LIN {X 0,Y 154.357,Z 466.364,A -85,B 0,C 180,E1 -24102.965,E2 -24102.965} C_VEL
LIN {X 0,Y 157.924,Z 467.612,A -85,B 0,C 180,E1 -24108.246,E2 -24108.246} C_VEL
LIN {X 0,Y 162.729,Z 467.187,A -85,B 0,C 180,E1 -24113.367,E2 -24113.367} C_VEL
LIN {X 0,Y 167.861,Z 465.471,A -85,B 0,C 180,E1 -24117.601,E2 -24117.601} C_VEL
LIN {X 0,Y 173.217,Z 462.762,A -85,B 0,C 180,E1 -24121.163,E2 -24121.163} C_VEL
LIN {X 0,Y 179.055,Z 458.948,A -85,B 0,C 180,E1 -24124.503,E2 -24124.503} C_VEL
LIN {X 0,Y 186.333,Z 453.105,A -85,B 0,C 180,E1 -24128.018,E2 -24128.018} C_VEL
LIN {X 0,Y 187.702,Z 451.908,A -85,B 0,C 180,E1 -24128.614,E2 -24128.614} C_VEL
LIN {X 0,Y 189.446,Z 450.085,A -85,B 0,C 180,E1 -24129.61,E2 -24129.61} C_VEL
LIN {X 0,Y 191.01,Z 446.938,A -85,B 0,C 180,E1 -24132.754,E2 -24132.754} C_VEL
LIN {X 0,Y 191.797,Z 445.035,A -85,B 0,C 180,E1 -24134.863,E2 -24134.863} C_VEL
LIN {X 0,Y 192.282,Z 443.477,A -85,B 0,C 180,E1 -24137.002,E2 -24137.002} C_VEL
LIN {X 0,Y 192.219,Z 442.595,A -85,B 0,C 180,E1 -24139.212,E2 -24139.212} C_VEL
LIN {X 0,Y 191.954,Z 442.263,A -85,B 0,C 180,E1 -24141.477,E2 -24141.477} C_VEL
LIN {X 0,Y 191.608,Z 442.354,A -85,B 0,C 180,E1 -24143.795,E2 -24143.795} C_VEL
LIN {X 0,Y 191.277,Z 442.94,A -85,B 0,C 180,E1 -24146.162,E2 -24146.162} C_VEL
LIN {X 0,Y 190.853,Z 444.09,A -85,B 0,C 180,E1 -24148.602,E2 -24148.602} C_VEL
LIN {X 0,Y 190.613,Z 447.54,A -85,B 0,C 180,E1 -24153.577,E2 -24153.577} C_VEL
LIN {X 0,Y 190.373,Z 450.298,A -85,B 0,C 180,E1 -24156.205,E2 -24156.205} C_VEL
LIN {X 0,Y 189.792,Z 454.164,A -85,B 0,C 180,E1 -24159.014,E2 -24159.014} C_VEL
LIN {X 0,Y 188.189,Z 457.579,A -85,B 0,C 180,E1 -24160.569,E2 -24160.569} C_VEL
LIN {X 0,Y 184.271,Z 464.734,A -85,B 0,C 180,E1 -24163.562,E2 -24163.562} C_VEL
LIN {X 0,Y 178.792,Z 473.353,A -85,B 0,C 180,E1 -24167.309,E2 -24167.309} C_VEL
LIN {X 0,Y 173.001,Z 480.936,A -85,B 0,C 180,E1 -24170.975,E2 -24170.975} C_VEL
LIN {X 0,Y 166.298,Z 488.194,A -85,B 0,C 180,E1 -24175.214,E2 -24175.214} C_VEL
LIN {X 0,Y 160.237,Z 493.898,A -85,B 0,C 180,E1 -24179.71,E2 -24179.71} C_VEL
LIN {X 0,Y 156.331,Z 497.231,A -85,B 0,C 180,E1 -24183.285,E2 -24183.285} C_VEL
LIN {X 0,Y 152.307,Z 500.47,A -85,B 0,C 180,E1 -24188.337,E2 -24188.337} C_VEL
LIN {X 0,Y 149.986,Z 502.425,A -85,B 0,C 180,E1 -24193.672,E2 -24193.672} C_VEL
LIN {X 0,Y 149.209,Z 503.02,A -85,B 0,C 180,E1 -24199.14,E2 -24199.14} C_VEL
LIN {X 0,Y 149.908,Z 502.28,A -85,B 0,C 180,E1 -24204.62,E2 -24204.62} C_VEL
LIN {X 0,Y 150.705,Z 501.363,A -85,B 0,C 180,E1 -24207.327,E2 -24207.327} C_VEL
LIN {X 0,Y 151.499,Z 500.007,A -85,B 0,C 180,E1 -24210,E2 -24210} C_VEL
LIN {X 0,Y 150.756,Z 496.519,A -85,B 0,C 180,E1 -24214.01,E2 -24214.01} C_VEL
LIN {X 0,Y 150.197,Z 491.756,A -85,B 0,C 180,E1 -24218.069,E2 -24218.069} C_VEL
LIN {X 0,Y 150.286,Z 485.644,A -85,B 0,C 180,E1 -24222.148,E2 -24222.148} C_VEL
LIN {X 0,Y 151,Z 477.97,A -85,B 0,C 180,E1 -24226.216,E2 -24226.216} C_VEL
LIN {X 0,Y 152.213,Z 470.164,A -85,B 0,C 180,E1 -24229.557,E2 -24229.557} C_VEL
LIN {X 0,Y 152.227,Z 462.309,A -85,B 0,C 180,E1 -24232.318,E2 -24232.318} C_VEL
LIN {X 0,Y 152.281,Z 452.364,A -85,B 0,C 180,E1 -24235.27,E2 -24235.27} C_VEL
LIN {X 0,Y 152.315,Z 441.552,A -85,B 0,C 180,E1 -24237.914,E2 -24237.914} C_VEL
LIN {X 0,Y 152.221,Z 428.27,A -85,B 0,C 180,E1 -24240.521,E2 -24240.521} C_VEL
LIN {X 0,Y 152.051,Z 415.268,A -85,B 0,C 180,E1 -24242.501,E2 -24242.501} C_VEL
LIN {X 0,Y 151.716,Z 401.613,A -85,B 0,C 180,E1 -24244.059,E2 -24244.059} C_VEL
LIN {X 0,Y 151.32,Z 399.501,A -85,B 0,C 180,E1 -24244.647,E2 -24244.647} C_VEL
LIN {X 0,Y 150.434,Z 397.793,A -85,B 0,C 180,E1 -24245.814,E2 -24245.814} C_VEL
LIN {X 0,Y 146.596,Z 391.678,A -85,B 0,C 180,E1 -24251.674,E2 -24251.674} C_VEL
LIN {X 0,Y 145.381,Z 388.003,A -85,B 0,C 180,E1 -24254.938,E2 -24254.938} C_VEL
LIN {X 0,Y 144.009,Z 381.533,A -85,B 0,C 180,E1 -24261.336,E2 -24261.336} C_VEL
LIN {X 0,Y 143.314,Z 377.702,A -85,B 0,C 180,E1 -24265.393,E2 -24265.393} C_VEL
LIN {X 0,Y 143.186,Z 377.647,A -85,B 0,C 180,E1 -24272.064,E2 -24272.064} C_VEL
LIN {X 0,Y 143.264,Z 377.634,A -85,B 0,C 180,E1 -24278.756,E2 -24278.756} C_VEL
LIN {X 0,Y 143.264,Z 377.64,A -85,B 0,C 180,E1 -24282.882,E2 -24282.882} C_VEL
LIN {X 0,Y 143.53,Z 377.598,A -85,B 0,C 180,E1 -24288.705,E2 -24288.705} C_VEL
LIN {X 0,Y 143.618,Z 377.594,A -85,B 0,C 180,E1 -24291.558,E2 -24291.558} C_VEL
LIN {X 0,Y 144.171,Z 377.525,A -85,B 0,C 180,E1 -24300,E2 -24300} C_VEL
LIN {X 0,Y 143.656,Z 377.59,A -85,B 0,C 180,E1 -24308.44,E2 -24308.44} C_VEL
LIN {X 0,Y 143.545,Z 377.601,A -85,B 0,C 180,E1 -24311.713,E2 -24311.713} C_VEL
LIN {X 0,Y 143.302,Z 377.634,A -85,B 0,C 180,E1 -24317.113,E2 -24317.113} C_VEL
LIN {X 0,Y 143.274,Z 377.632,A -85,B 0,C 180,E1 -24321.255,E2 -24321.255} C_VEL
LIN {X 0,Y 143.188,Z 377.648,A -85,B 0,C 180,E1 -24327.938,E2 -24327.938} C_VEL
LIN {X 0,Y 143.167,Z 377.65,A -85,B 0,C 180,E1 -24333.436,E2 -24333.436} C_VEL
LIN {X 0,Y 143.077,Z 377.659,A -85,B 0,C 180,E1 -24339.685,E2 -24339.685} C_VEL
LIN {X 0,Y 143.066,Z 377.663,A -85,B 0,C 180,E1 -24343.451,E2 -24343.451} C_VEL
LIN {X 0,Y 143.069,Z 377.659,A -85,B 0,C 180,E1 -24347.464,E2 -24347.464} C_VEL
LIN {X 0,Y 143.106,Z 377.659,A -85,B 0,C 180,E1 -24351.792,E2 -24351.792} C_VEL
LIN {X 0,Y 143.185,Z 377.647,A -85,B 0,C 180,E1 -24357.323,E2 -24357.323} C_VEL
LIN {X 0,Y 143.191,Z 377.644,A -85,B 0,C 180,E1 -24362.063,E2 -24362.063} C_VEL
LIN {X 0,Y 143.278,Z 377.636,A -85,B 0,C 180,E1 -24368.746,E2 -24368.746} C_VEL
LIN {X 0,Y 143.318,Z 377.629,A -85,B 0,C 180,E1 -24372.889,E2 -24372.889} C_VEL
LIN {X 0,Y 143.604,Z 377.592,A -85,B 0,C 180,E1 -24378.711,E2 -24378.711} C_VEL
LIN {X 0,Y 143.687,Z 377.585,A -85,B 0,C 180,E1 -24381.562,E2 -24381.562} C_VEL
LIN {X 0,Y 144.18,Z 377.526,A -85,B 0,C 180,E1 -24390,E2 -24390} C_VEL
LIN {X 0,Y 143.662,Z 377.589,A -85,B 0,C 180,E1 -24398.439,E2 -24398.439} C_VEL
LIN {X 0,Y 143.549,Z 377.598,A -85,B 0,C 180,E1 -24401.712,E2 -24401.712} C_VEL
LIN {X 0,Y 143.309,Z 377.631,A -85,B 0,C 180,E1 -24407.112,E2 -24407.112} C_VEL
LIN {X 0,Y 143.279,Z 377.636,A -85,B 0,C 180,E1 -24411.255,E2 -24411.255} C_VEL
LIN {X 0,Y 143.204,Z 377.646,A -85,B 0,C 180,E1 -24418.433,E2 -24418.433} C_VEL
LIN {X 0,Y 143.215,Z 377.783,A -85,B 0,C 180,E1 -24419.148,E2 -24419.148} C_VEL
LIN {X 0,Y 143.551,Z 379.072,A -85,B 0,C 180,E1 -24419.715,E2 -24419.715} C_VEL
LIN {X 0,Y 147.266,Z 391.351,A -85,B 0,C 180,E1 -24422.471,E2 -24422.471} C_VEL
LIN {X 0,Y 150.191,Z 402.477,A -85,B 0,C 180,E1 -24425.295,E2 -24425.295} C_VEL
LIN {X 0,Y 151.278,Z 407.074,A -85,B 0,C 180,E1 -24426.585,E2 -24426.585} C_VEL
LIN {X 0,Y 150.775,Z 410.846,A -85,B 0,C 180,E1 -24427.589,E2 -24427.589} C_VEL
LIN {X 0,Y 148.66,Z 421.695,A -85,B 0,C 180,E1 -24430.851,E2 -24430.851} C_VEL
LIN {X 0,Y 146.664,Z 431.947,A -85,B 0,C 180,E1 -24434.715,E2 -24434.715} C_VEL
LIN {X 0,Y 145.272,Z 439.714,A -85,B 0,C 180,E1 -24438.302,E2 -24438.302} C_VEL
LIN {X 0,Y 144.152,Z 447.331,A -85,B 0,C 180,E1 -24442.593,E2 -24442.593} C_VEL
LIN {X 0,Y 143.579,Z 454.147,A -85,B 0,C 180,E1 -24447.423,E2 -24447.423} C_VEL
LIN {X 0,Y 143.684,Z 458.94,A -85,B 0,C 180,E1 -24451.692,E2 -24451.692} C_VEL
LIN {X 0,Y 144.77,Z 463.725,A -85,B 0,C 180,E1 -24457.272,E2 -24457.272} C_VEL
LIN {X 0,Y 147.105,Z 466.924,A -85,B 0,C 180,E1 -24462.84,E2 -24462.84} C_VEL
LIN {X 0,Y 150.694,Z 468.63,A -85,B 0,C 180,E1 -24468.34,E2 -24468.34} C_VEL
LIN {X 0,Y 155.575,Z 468.704,A -85,B 0,C 180,E1 -24473.621,E2 -24473.621} C_VEL
LIN {X 0,Y 161.684,Z 467.121,A -85,B 0,C 180,E1 -24478.668,E2 -24478.668} C_VEL
LIN {X 0,Y 168.951,Z 463.815,A -85,B 0,C 180,E1 -24483.318,E2 -24483.318} C_VEL
LIN {X 0,Y 175.778,Z 459.555,A -85,B 0,C 180,E1 -24486.889,E2 -24486.889} C_VEL
LIN {X 0,Y 182.642,Z 454.306,A -85,B 0,C 180,E1 -24489.972,E2 -24489.972} C_VEL
LIN {X 0,Y 184.158,Z 452.844,A -85,B 0,C 180,E1 -24491,E2 -24491} C_VEL
LIN {X 0,Y 185.308,Z 451.011,A -85,B 0,C 180,E1 -24493.153,E2 -24493.153} C_VEL
LIN {X 0,Y 186.297,Z 449.275,A -85,B 0,C 180,E1 -24495.312,E2 -24495.312} C_VEL
LIN {X 0,Y 186.916,Z 447.95,A -85,B 0,C 180,E1 -24497.506,E2 -24497.506} C_VEL
LIN {X 0,Y 186.882,Z 447.289,A -85,B 0,C 180,E1 -24499.925,E2 -24499.925} C_VEL
LIN {X 0,Y 186.707,Z 447.179,A -85,B 0,C 180,E1 -24502.112,E2 -24502.112} C_VEL
LIN {X 0,Y 186.317,Z 447.696,A -85,B 0,C 180,E1 -24505.14,E2 -24505.14} C_VEL
LIN {X 0,Y 186.072,Z 448.315,A -85,B 0,C 180,E1 -24506.952,E2 -24506.952} C_VEL
LIN {X 0,Y 185.445,Z 451.37,A -85,B 0,C 180,E1 -24512.044,E2 -24512.044} C_VEL
LIN {X 0,Y 185.308,Z 453.622,A -85,B 0,C 180,E1 -24514.673,E2 -24514.673} C_VEL
LIN {X 0,Y 184.592,Z 457.005,A -85,B 0,C 180,E1 -24517.53,E2 -24517.53} C_VEL
LIN {X 0,Y 184.039,Z 458.562,A -85,B 0,C 180,E1 -24518.509,E2 -24518.509} C_VEL
LIN {X 0,Y 179.381,Z 465.993,A -85,B 0,C 180,E1 -24521.894,E2 -24521.894} C_VEL
LIN {X 0,Y 174.417,Z 473.037,A -85,B 0,C 180,E1 -24525.16,E2 -24525.16} C_VEL
LIN {X 0,Y 169.27,Z 479.371,A -85,B 0,C 180,E1 -24528.372,E2 -24528.372} C_VEL
LIN {X 0,Y 163.931,Z 484.915,A -85,B 0,C 180,E1 -24531.565,E2 -24531.565} C_VEL
LIN {X 0,Y 157.251,Z 491.061,A -85,B 0,C 180,E1 -24536.038,E2 -24536.038} C_VEL
LIN {X 0,Y 152.664,Z 494.674,A -85,B 0,C 180,E1 -24539.577,E2 -24539.577} C_VEL
LIN {X 0,Y 147.621,Z 498.32,A -85,B 0,C 180,E1 -24544.63,E2 -24544.63} C_VEL
LIN {X 0,Y 144.256,Z 500.64,A -85,B 0,C 180,E1 -24550.061,E2 -24550.061} C_VEL
LIN {X 0,Y 142.518,Z 501.685,A -85,B 0,C 180,E1 -24555.726,E2 -24555.726} C_VEL
LIN {X 0,Y 142.435,Z 501.436,A -85,B 0,C 180,E1 -24561.488,E2 -24561.488} C_VEL
LIN {X 0,Y 143.727,Z 499.805,A -85,B 0,C 180,E1 -24567.197,E2 -24567.197} C_VEL
LIN {X 0,Y 144.54,Z 498.311,A -85,B 0,C 180,E1 -24570,E2 -24570} C_VEL
LIN {X 0,Y 143.749,Z 494.605,A -85,B 0,C 180,E1 -24574.206,E2 -24574.206} C_VEL
LIN {X 0,Y 143.219,Z 489.598,A -85,B 0,C 180,E1 -24578.465,E2 -24578.465} C_VEL
LIN {X 0,Y 143.379,Z 483.237,A -85,B 0,C 180,E1 -24582.743,E2 -24582.743} C_VEL
LIN {X 0,Y 144.239,Z 475.28,A -85,B 0,C 180,E1 -24586.998,E2 -24586.998} C_VEL
LIN {X 0,Y 145.174,Z 468.85,A -85,B 0,C 180,E1 -24589.808,E2 -24589.808} C_VEL
LIN {X 0,Y 145.165,Z 459.805,A -85,B 0,C 180,E1 -24593.093,E2 -24593.093} C_VEL
LIN {X 0,Y 145.254,Z 448,A -85,B 0,C 180,E1 -24596.586,E2 -24596.586} C_VEL
LIN {X 0,Y 145.302,Z 435.99,A -85,B 0,C 180,E1 -24599.468,E2 -24599.468} C_VEL
LIN {X 0,Y 145.193,Z 422.691,A -85,B 0,C 180,E1 -24601.982,E2 -24601.982} C_VEL
LIN {X 0,Y 145.003,Z 408.799,A -85,B 0,C 180,E1 -24603.987,E2 -24603.987} C_VEL
LIN {X 0,Y 144.923,Z 398.818,A -85,B 0,C 180,E1 -24605.188,E2 -24605.188} C_VEL
LIN {X 0,Y 146.169,Z 394.703,A -85,B 0,C 180,E1 -24608.685,E2 -24608.685} C_VEL
LIN {X 0,Y 146.437,Z 392.265,A -85,B 0,C 180,E1 -24610.919,E2 -24610.919} C_VEL
LIN {X 0,Y 145.381,Z 388.003,A -85,B 0,C 180,E1 -24614.938,E2 -24614.938} C_VEL
LIN {X 0,Y 144.38,Z 386.609,A -85,B 0,C 180,E1 -24616.344,E2 -24616.344} C_VEL
LIN {X 0,Y 141.069,Z 384.674,A -85,B 0,C 180,E1 -24618.55,E2 -24618.55} C_VEL
LIN {X 0,Y 137.744,Z 382.744,A -85,B 0,C 180,E1 -24620.858,E2 -24620.858} C_VEL
LIN {X 0,Y 136.779,Z 381.393,A -85,B 0,C 180,E1 -24622.388,E2 -24622.388} C_VEL
LIN {X 0,Y 136.26,Z 378.572,A -85,B 0,C 180,E1 -24625.611,E2 -24625.611} C_VEL
LIN {X 0,Y 136.142,Z 378.524,A -85,B 0,C 180,E1 -24632.315,E2 -24632.315} C_VEL
LIN {X 0,Y 136.231,Z 378.51,A -85,B 0,C 180,E1 -24638.831,E2 -24638.831} C_VEL
LIN {X 0,Y 136.23,Z 378.508,A -85,B 0,C 180,E1 -24645.052,E2 -24645.052} C_VEL
LIN {X 0,Y 136.423,Z 378.482,A -85,B 0,C 180,E1 -24648.177,E2 -24648.177} C_VEL
LIN {X 0,Y 136.544,Z 378.476,A -85,B 0,C 180,E1 -24651.117,E2 -24651.117} C_VEL
LIN {X 0,Y 137.128,Z 378.402,A -85,B 0,C 180,E1 -24660,E2 -24660} C_VEL
LIN {X 0,Y 136.584,Z 378.472,A -85,B 0,C 180,E1 -24668.88,E2 -24668.88} C_VEL
LIN {X 0,Y 136.489,Z 378.481,A -85,B 0,C 180,E1 -24671.955,E2 -24671.955} C_VEL
LIN {X 0,Y 136.241,Z 378.514,A -85,B 0,C 180,E1 -24678.03,E2 -24678.03} C_VEL
LIN {X 0,Y 136.195,Z 378.513,A -85,B 0,C 180,E1 -24681.749,E2 -24681.749} C_VEL
LIN {X 0,Y 136.098,Z 378.528,A -85,B 0,C 180,E1 -24688.617,E2 -24688.617} C_VEL
LIN {X 0,Y 136.077,Z 378.534,A -85,B 0,C 180,E1 -24694.619,E2 -24694.619} C_VEL
LIN {X 0,Y 136.052,Z 378.533,A -85,B 0,C 180,E1 -24699.21,E2 -24699.21} C_VEL
LIN {X 0,Y 136.006,Z 378.543,A -85,B 0,C 180,E1 -24703.662,E2 -24703.662} C_VEL
LIN {X 0,Y 136.033,Z 378.536,A -85,B 0,C 180,E1 -24707.808,E2 -24707.808} C_VEL
LIN {X 0,Y 136.055,Z 378.537,A -85,B 0,C 180,E1 -24711.695,E2 -24711.695} C_VEL
LIN {X 0,Y 136.09,Z 378.528,A -85,B 0,C 180,E1 -24715.718,E2 -24715.718} C_VEL
LIN {X 0,Y 136.147,Z 378.52,A -85,B 0,C 180,E1 -24722.317,E2 -24722.317} C_VEL
LIN {X 0,Y 136.245,Z 378.512,A -85,B 0,C 180,E1 -24728.834,E2 -24728.834} C_VEL
LIN {X 0,Y 136.287,Z 378.508,A -85,B 0,C 180,E1 -24735.059,E2 -24735.059} C_VEL
LIN {X 0,Y 136.502,Z 378.477,A -85,B 0,C 180,E1 -24738.115,E2 -24738.115} C_VEL
LIN {X 0,Y 136.61,Z 378.464,A -85,B 0,C 180,E1 -24741.122,E2 -24741.122} C_VEL
LIN {X 0,Y 137.137,Z 378.403,A -85,B 0,C 180,E1 -24750,E2 -24750} C_VEL
LIN {X 0,Y 136.59,Z 378.471,A -85,B 0,C 180,E1 -24758.879,E2 -24758.879} C_VEL
LIN {X 0,Y 136.492,Z 378.476,A -85,B 0,C 180,E1 -24761.954,E2 -24761.954} C_VEL
LIN {X 0,Y 136.248,Z 378.513,A -85,B 0,C 180,E1 -24768.028,E2 -24768.028} C_VEL
LIN {X 0,Y 136.2,Z 378.519,A -85,B 0,C 180,E1 -24771.749,E2 -24771.749} C_VEL
LIN {X 0,Y 136.215,Z 378.742,A -85,B 0,C 180,E1 -24778.366,E2 -24778.366} C_VEL
LIN {X 0,Y 136.564,Z 380.219,A -85,B 0,C 180,E1 -24778.952,E2 -24778.952} C_VEL
LIN {X 0,Y 140.044,Z 391.581,A -85,B 0,C 180,E1 -24781.629,E2 -24781.629} C_VEL
LIN {X 0,Y 142.86,Z 402.224,A -85,B 0,C 180,E1 -24784.453,E2 -24784.453} C_VEL
LIN {X 0,Y 144.294,Z 408.184,A -85,B 0,C 180,E1 -24786.195,E2 -24786.195} C_VEL
LIN {X 0,Y 142.369,Z 418.599,A -85,B 0,C 180,E1 -24789.244,E2 -24789.244} C_VEL
LIN {X 0,Y 140.108,Z 429.837,A -85,B 0,C 180,E1 -24793.338,E2 -24793.338} C_VEL
LIN {X 0,Y 138.322,Z 439.282,A -85,B 0,C 180,E1 -24797.684,E2 -24797.684} C_VEL
LIN {X 0,Y 137.152,Z 446.946,A -85,B 0,C 180,E1 -24802.055,E2 -24802.055} C_VEL
LIN {X 0,Y 136.487,Z 454.243,A -85,B 0,C 180,E1 -24807.271,E2 -24807.271} C_VEL
LIN {X 0,Y 136.663,Z 459.872,A -85,B 0,C 180,E1 -24812.43,E2 -24812.43} C_VEL
LIN {X 0,Y 137.548,Z 463.697,A -85,B 0,C 180,E1 -24816.88,E2 -24816.88} C_VEL
LIN {X 0,Y 139.85,Z 467.374,A -85,B 0,C 180,E1 -24822.707,E2 -24822.707} C_VEL
LIN {X 0,Y 143.461,Z 469.494,A -85,B 0,C 180,E1 -24828.45,E2 -24828.45} C_VEL
LIN {X 0,Y 146.201,Z 470.045,A -85,B 0,C 180,E1 -24831.708,E2 -24831.708} C_VEL
LIN {X 0,Y 149.094,Z 470.03,A -85,B 0,C 180,E1 -24834.59,E2 -24834.59} C_VEL
LIN {X 0,Y 154.629,Z 469.025,A -85,B 0,C 180,E1 -24839.143,E2 -24839.143} C_VEL
LIN {X 0,Y 162.013,Z 466.324,A -85,B 0,C 180,E1 -24843.888,E2 -24843.888} C_VEL
LIN {X 0,Y 168.225,Z 463.079,A -85,B 0,C 180,E1 -24847.2,E2 -24847.2} C_VEL
LIN {X 0,Y 175.256,Z 458.564,A -85,B 0,C 180,E1 -24850.396,E2 -24850.396} C_VEL
LIN {X 0,Y 177.687,Z 456.802,A -85,B 0,C 180,E1 -24851.406,E2 -24851.406} C_VEL
LIN {X 0,Y 179.485,Z 454.864,A -85,B 0,C 180,E1 -24853.588,E2 -24853.588} C_VEL
LIN {X 0,Y 180.701,Z 453.339,A -85,B 0,C 180,E1 -24855.798,E2 -24855.798} C_VEL
LIN {X 0,Y 181.365,Z 452.239,A -85,B 0,C 180,E1 -24858.06,E2 -24858.06} C_VEL
LIN {X 0,Y 181.364,Z 451.826,A -85,B 0,C 180,E1 -24861.566,E2 -24861.566} C_VEL
LIN {X 0,Y 180.963,Z 452.486,A -85,B 0,C 180,E1 -24865.29,E2 -24865.29} C_VEL
LIN {X 0,Y 180.506,Z 453.579,A -85,B 0,C 180,E1 -24867.854,E2 -24867.854} C_VEL
LIN {X 0,Y 180.026,Z 456.917,A -85,B 0,C 180,E1 -24873.13,E2 -24873.13} C_VEL
LIN {X 0,Y 179.314,Z 459.81,A -85,B 0,C 180,E1 -24876.009,E2 -24876.009} C_VEL
LIN {X 0,Y 178.876,Z 461.072,A -85,B 0,C 180,E1 -24877.004,E2 -24877.004} C_VEL
LIN {X 0,Y 177.22,Z 463.734,A -85,B 0,C 180,E1 -24878.446,E2 -24878.446} C_VEL
LIN {X 0,Y 172.055,Z 470.575,A -85,B 0,C 180,E1 -24881.802,E2 -24881.802} C_VEL
LIN {X 0,Y 165.796,Z 477.898,A -85,B 0,C 180,E1 -24885.621,E2 -24885.621} C_VEL
LIN {X 0,Y 160.266,Z 483.373,A -85,B 0,C 180,E1 -24888.87,E2 -24888.87} C_VEL
LIN {X 0,Y 153.015,Z 489.519,A -85,B 0,C 180,E1 -24893.339,E2 -24893.339} C_VEL
LIN {X 0,Y 146.557,Z 494.203,A -85,B 0,C 180,E1 -24898.165,E2 -24898.165} C_VEL
LIN {X 0,Y 141.21,Z 497.544,A -85,B 0,C 180,E1 -24903.39,E2 -24903.39} C_VEL
LIN {X 0,Y 137.573,Z 499.634,A -85,B 0,C 180,E1 -24909.048,E2 -24909.048} C_VEL
LIN {X 0,Y 135.637,Z 500.465,A -85,B 0,C 180,E1 -24914.985,E2 -24914.985} C_VEL
LIN {X 0,Y 135.44,Z 499.99,A -85,B 0,C 180,E1 -24921.045,E2 -24921.045} C_VEL
LIN {X 0,Y 136.769,Z 498.123,A -85,B 0,C 180,E1 -24927.055,E2 -24927.055} C_VEL
LIN {X 0,Y 137.592,Z 496.559,A -85,B 0,C 180,E1 -24930,E2 -24930} C_VEL
LIN {X 0,Y 136.729,Z 492.653,A -85,B 0,C 180,E1 -24934.422,E2 -24934.422} C_VEL
LIN {X 0,Y 136.239,Z 487.441,A -85,B 0,C 180,E1 -24938.903,E2 -24938.903} C_VEL
LIN {X 0,Y 136.45,Z 480.782,A -85,B 0,C 180,E1 -24943.401,E2 -24943.401} C_VEL
LIN {X 0,Y 137.524,Z 472.475,A -85,B 0,C 180,E1 -24947.855,E2 -24947.855} C_VEL
LIN {X 0,Y 138.132,Z 467.508,A -85,B 0,C 180,E1 -24950.086,E2 -24950.086} C_VEL
LIN {X 0,Y 138.079,Z 456.924,A -85,B 0,C 180,E1 -24954.028,E2 -24954.028} C_VEL
LIN {X 0,Y 138.187,Z 444.955,A -85,B 0,C 180,E1 -24957.65,E2 -24957.65} C_VEL
LIN {X 0,Y 138.258,Z 432.958,A -85,B 0,C 180,E1 -24960.551,E2 -24960.551} C_VEL
LIN {X 0,Y 138.262,Z 419.62,A -85,B 0,C 180,E1 -24963.122,E2 -24963.122} C_VEL
LIN {X 0,Y 138.102,Z 405.043,A -85,B 0,C 180,E1 -24965.212,E2 -24965.212} C_VEL
LIN {X 0,Y 138.081,Z 397.764,A -85,B 0,C 180,E1 -24966.14,E2 -24966.14} C_VEL
LIN {X 0,Y 139.151,Z 394.496,A -85,B 0,C 180,E1 -24969.086,E2 -24969.086} C_VEL
LIN {X 0,Y 139.317,Z 392.541,A -85,B 0,C 180,E1 -24970.979,E2 -24970.979} C_VEL
LIN {X 0,Y 137.852,Z 386.623,A -85,B 0,C 180,E1 -24976.893,E2 -24976.893} C_VEL
LIN {X 0,Y 136.779,Z 381.393,A -85,B 0,C 180,E1 -24982.388,E2 -24982.388} C_VEL
LIN {X 0,Y 136.203,Z 380.228,A -85,B 0,C 180,E1 -24983.939,E2 -24983.939} C_VEL
LIN {X 0,Y 134.584,Z 379.264,A -85,B 0,C 180,E1 -24986.31,E2 -24986.31} C_VEL
LIN {X 0,Y 132.573,Z 378.987,A -85,B 0,C 180,E1 -24988.714,E2 -24988.714} C_VEL
LIN {X 0,Y 129.287,Z 379.385,A -85,B 0,C 180,E1 -24993.846,E2 -24993.846} C_VEL
LIN {X 0,Y 129.002,Z 379.405,A -85,B 0,C 180,E1 -24995.637,E2 -24995.637} C_VEL
LIN {X 0,Y 129.111,Z 379.402,A -85,B 0,C 180,E1 -25000.937,E2 -25000.937} C_VEL
LIN {X 0,Y 129.341,Z 379.364,A -85,B 0,C 180,E1 -25007.97,E2 -25007.97} C_VEL
LIN {X 0,Y 129.467,Z 379.355,A -85,B 0,C 180,E1 -25010.627,E2 -25010.627} C_VEL
LIN {X 0,Y 130.083,Z 379.28,A -85,B 0,C 180,E1 -25020,E2 -25020} C_VEL
LIN {X 0,Y 129.511,Z 379.352,A -85,B 0,C 180,E1 -25029.369,E2 -25029.369} C_VEL
LIN {X 0,Y 129.39,Z 379.363,A -85,B 0,C 180,E1 -25032.548,E2 -25032.548} C_VEL
LIN {X 0,Y 129.152,Z 379.396,A -85,B 0,C 180,E1 -25039.056,E2 -25039.056} C_VEL
LIN {X 0,Y 129.106,Z 379.397,A -85,B 0,C 180,E1 -25042.399,E2 -25042.399} C_VEL
LIN {X 0,Y 129.034,Z 379.406,A -85,B 0,C 180,E1 -25049.374,E2 -25049.374} C_VEL
LIN {X 0,Y 128.991,Z 379.416,A -85,B 0,C 180,E1 -25055.19,E2 -25055.19} C_VEL
LIN {X 0,Y 128.975,Z 379.418,A -85,B 0,C 180,E1 -25060.836,E2 -25060.836} C_VEL
LIN {X 0,Y 128.924,Z 379.422,A -85,B 0,C 180,E1 -25065.126,E2 -25065.126} C_VEL
LIN {X 0,Y 128.957,Z 379.421,A -85,B 0,C 180,E1 -25069.728,E2 -25069.728} C_VEL
LIN {X 0,Y 128.991,Z 379.411,A -85,B 0,C 180,E1 -25074.812,E2 -25074.812} C_VEL
LIN {X 0,Y 129.051,Z 379.408,A -85,B 0,C 180,E1 -25080.652,E2 -25080.652} C_VEL
LIN {X 0,Y 129.108,Z 379.404,A -85,B 0,C 180,E1 -25087.728,E2 -25087.728} C_VEL
LIN {X 0,Y 129.161,Z 379.39,A -85,B 0,C 180,E1 -25090.945,E2 -25090.945} C_VEL
LIN {X 0,Y 129.42,Z 379.361,A -85,B 0,C 180,E1 -25097.816,E2 -25097.816} C_VEL
LIN {X 0,Y 129.532,Z 379.345,A -85,B 0,C 180,E1 -25100.633,E2 -25100.633} C_VEL
LIN {X 0,Y 130.092,Z 379.281,A -85,B 0,C 180,E1 -25110,E2 -25110} C_VEL
LIN {X 0,Y 129.516,Z 379.353,A -85,B 0,C 180,E1 -25119.369,E2 -25119.369} C_VEL
LIN {X 0,Y 129.394,Z 379.361,A -85,B 0,C 180,E1 -25122.548,E2 -25122.548} C_VEL
LIN {X 0,Y 129.158,Z 379.398,A -85,B 0,C 180,E1 -25129.055,E2 -25129.055} C_VEL
LIN {X 0,Y 129.109,Z 379.403,A -85,B 0,C 180,E1 -25132.398,E2 -25132.398} C_VEL
LIN {X 0,Y 129.111,Z 379.513,A -85,B 0,C 180,E1 -25137.34,E2 -25137.34} C_VEL
LIN {X 0,Y 129.362,Z 380.61,A -85,B 0,C 180,E1 -25137.942,E2 -25137.942} C_VEL
LIN {X 0,Y 132.87,Z 392.094,A -85,B 0,C 180,E1 -25140.777,E2 -25140.777} C_VEL
LIN {X 0,Y 135.839,Z 403.192,A -85,B 0,C 180,E1 -25143.881,E2 -25143.881} C_VEL
LIN {X 0,Y 137.231,Z 408.847,A -85,B 0,C 180,E1 -25145.629,E2 -25145.629} C_VEL
LIN {X 0,Y 135.513,Z 418.313,A -85,B 0,C 180,E1 -25148.487,E2 -25148.487} C_VEL
LIN {X 0,Y 133.301,Z 428.928,A -85,B 0,C 180,E1 -25152.429,E2 -25152.429} C_VEL
LIN {X 0,Y 131.445,Z 438.503,A -85,B 0,C 180,E1 -25156.885,E2 -25156.885} C_VEL
LIN {X 0,Y 130.136,Z 446.657,A -85,B 0,C 180,E1 -25161.607,E2 -25161.607} C_VEL
LIN {X 0,Y 129.396,Z 454.227,A -85,B 0,C 180,E1 -25167.102,E2 -25167.102} C_VEL
LIN {X 0,Y 129.598,Z 460.172,A -85,B 0,C 180,E1 -25172.552,E2 -25172.552} C_VEL
LIN {X 0,Y 130.703,Z 464.645,A -85,B 0,C 180,E1 -25177.889,E2 -25177.889} C_VEL
LIN {X 0,Y 132.578,Z 467.655,A -85,B 0,C 180,E1 -25182.585,E2 -25182.585} C_VEL
LIN {X 0,Y 136.224,Z 470.238,A -85,B 0,C 180,E1 -25188.582,E2 -25188.582} C_VEL
LIN {X 0,Y 138.346,Z 470.922,A -85,B 0,C 180,E1 -25191.234,E2 -25191.234} C_VEL
LIN {X 0,Y 141.253,Z 471.297,A -85,B 0,C 180,E1 -25194.309,E2 -25194.309} C_VEL
LIN {X 0,Y 147.586,Z 470.778,A -85,B 0,C 180,E1 -25199.694,E2 -25199.694} C_VEL
LIN {X 0,Y 155.102,Z 468.626,A -85,B 0,C 180,E1 -25204.557,E2 -25204.557} C_VEL
LIN {X 0,Y 160.575,Z 466.351,A -85,B 0,C 180,E1 -25207.545,E2 -25207.545} C_VEL
LIN {X 0,Y 167.851,Z 462.44,A -85,B 0,C 180,E1 -25210.861,E2 -25210.861} C_VEL
LIN {X 0,Y 172.473,Z 459.413,A -85,B 0,C 180,E1 -25212.951,E2 -25212.951} C_VEL
LIN {X 0,Y 173.501,Z 458.564,A -85,B 0,C 180,E1 -25214.066,E2 -25214.066} C_VEL
LIN {X 0,Y 174.968,Z 457.191,A -85,B 0,C 180,E1 -25216.33,E2 -25216.33} C_VEL
LIN {X 0,Y 175.649,Z 456.336,A -85,B 0,C 180,E1 -25218.669,E2 -25218.669} C_VEL
LIN {X 0,Y 175.803,Z 456.179,A -85,B 0,C 180,E1 -25221.087,E2 -25221.087} C_VEL
LIN {X 0,Y 175.516,Z 456.527,A -85,B 0,C 180,E1 -25223.605,E2 -25223.605} C_VEL
LIN {X 0,Y 175.288,Z 457.266,A -85,B 0,C 180,E1 -25226.17,E2 -25226.17} C_VEL
LIN {X 0,Y 174.39,Z 460.669,A -85,B 0,C 180,E1 -25232.19,E2 -25232.19} C_VEL
LIN {X 0,Y 173.947,Z 462.597,A -85,B 0,C 180,E1 -25234.447,E2 -25234.447} C_VEL
LIN {X 0,Y 173.375,Z 464.096,A -85,B 0,C 180,E1 -25235.835,E2 -25235.835} C_VEL
LIN {X 0,Y 172.76,Z 465.1,A -85,B 0,C 180,E1 -25236.542,E2 -25236.542} C_VEL
LIN {X 0,Y 167.757,Z 471.028,A -85,B 0,C 180,E1 -25239.691,E2 -25239.691} C_VEL
LIN {X 0,Y 160.732,Z 478.381,A -85,B 0,C 180,E1 -25243.826,E2 -25243.826} C_VEL
LIN {X 0,Y 154.939,Z 483.579,A -85,B 0,C 180,E1 -25247.127,E2 -25247.127} C_VEL
LIN {X 0,Y 147.332,Z 489.304,A -85,B 0,C 180,E1 -25251.676,E2 -25251.676} C_VEL
LIN {X 0,Y 140.557,Z 493.694,A -85,B 0,C 180,E1 -25256.633,E2 -25256.633} C_VEL
LIN {X 0,Y 134.881,Z 496.778,A -85,B 0,C 180,E1 -25262.035,E2 -25262.035} C_VEL
LIN {X 0,Y 130.941,Z 498.583,A -85,B 0,C 180,E1 -25267.932,E2 -25267.932} C_VEL
LIN {X 0,Y 128.807,Z 499.152,A -85,B 0,C 180,E1 -25274.169,E2 -25274.169} C_VEL
LIN {X 0,Y 128.483,Z 498.47,A -85,B 0,C 180,E1 -25280.555,E2 -25280.555} C_VEL
LIN {X 0,Y 129.799,Z 496.447,A -85,B 0,C 180,E1 -25286.896,E2 -25286.896} C_VEL
LIN {X 0,Y 130.652,Z 494.75,A -85,B 0,C 180,E1 -25290,E2 -25290} C_VEL
LIN {X 0,Y 129.717,Z 490.585,A -85,B 0,C 180,E1 -25294.661,E2 -25294.661} C_VEL
LIN {X 0,Y 129.335,Z 483.917,A -85,B 0,C 180,E1 -25300.289,E2 -25300.289} C_VEL
LIN {X 0,Y 129.734,Z 476.887,A -85,B 0,C 180,E1 -25304.911,E2 -25304.911} C_VEL
LIN {X 0,Y 131.014,Z 467.886,A -85,B 0,C 180,E1 -25309.588,E2 -25309.588} C_VEL
LIN {X 0,Y 131.012,Z 458.674,A -85,B 0,C 180,E1 -25313.377,E2 -25313.377} C_VEL
LIN {X 0,Y 131.107,Z 447.608,A -85,B 0,C 180,E1 -25317.105,E2 -25317.105} C_VEL
LIN {X 0,Y 131.235,Z 436.153,A -85,B 0,C 180,E1 -25320.243,E2 -25320.243} C_VEL
LIN {X 0,Y 131.282,Z 423.415,A -85,B 0,C 180,E1 -25323.049,E2 -25323.049} C_VEL
LIN {X 0,Y 131.258,Z 409.622,A -85,B 0,C 180,E1 -25325.375,E2 -25325.375} C_VEL
LIN {X 0,Y 131.229,Z 396.947,A -85,B 0,C 180,E1 -25327.068,E2 -25327.068} C_VEL
LIN {X 0,Y 132.112,Z 394.088,A -85,B 0,C 180,E1 -25329.669,E2 -25329.669} C_VEL
LIN {X 0,Y 131.992,Z 392.014,A -85,B 0,C 180,E1 -25331.803,E2 -25331.803} C_VEL
LIN {X 0,Y 130.636,Z 386.584,A -85,B 0,C 180,E1 -25337.554,E2 -25337.554} C_VEL
LIN {X 0,Y 129.584,Z 381.372,A -85,B 0,C 180,E1 -25343.374,E2 -25343.374} C_VEL
LIN {X 0,Y 129.186,Z 379.445,A -85,B 0,C 180,E1 -25345.785,E2 -25345.785} C_VEL
LIN {X 0,Y 129.049,Z 379.406,A -85,B 0,C 180,E1 -25350.65,E2 -25350.65} C_VEL
LIN {X 0,Y 129.002,Z 379.405,A -85,B 0,C 180,E1 -25355.637,E2 -25355.637} C_VEL
LIN {X 0,Y 128.367,Z 379.489,A -85,B 0,C 180,E1 -25358.242,E2 -25358.242} C_VEL
LIN {X 0,Y 126.825,Z 379.687,A -85,B 0,C 180,E1 -25360.816,E2 -25360.816} C_VEL
LIN {X 0,Y 122.549,Z 380.209,A -85,B 0,C 180,E1 -25367.937,E2 -25367.937} C_VEL
LIN {X 0,Y 122.37,Z 380.236,A -85,B 0,C 180,E1 -25369.814,E2 -25369.814} C_VEL
LIN {X 0,Y 122.588,Z 380.209,A -85,B 0,C 180,E1 -25376.713,E2 -25376.713} C_VEL
LIN {X 0,Y 123.036,Z 380.158,A -85,B 0,C 180,E1 -25380,E2 -25380} C_VEL
LIN {X 0,Y 122.409,Z 380.23,A -85,B 0,C 180,E1 -25387.18,E2 -25387.18} C_VEL
LIN {X 0,Y 122.361,Z 380.238,A -85,B 0,C 180,E1 -25392.473,E2 -25392.473} C_VEL
LIN {X 0,Y 122.044,Z 380.28,A -85,B 0,C 180,E1 -25400.213,E2 -25400.213} C_VEL
LIN {X 0,Y 121.981,Z 380.288,A -85,B 0,C 180,E1 -25403.785,E2 -25403.785} C_VEL
LIN {X 0,Y 121.94,Z 380.29,A -85,B 0,C 180,E1 -25410.174,E2 -25410.174} C_VEL
LIN {X 0,Y 121.912,Z 380.297,A -85,B 0,C 180,E1 -25416.191,E2 -25416.191} C_VEL
LIN {X 0,Y 121.902,Z 380.299,A -85,B 0,C 180,E1 -25421.456,E2 -25421.456} C_VEL
LIN {X 0,Y 121.884,Z 380.302,A -85,B 0,C 180,E1 -25428.555,E2 -25428.555} C_VEL
LIN {X 0,Y 121.944,Z 380.288,A -85,B 0,C 180,E1 -25434.808,E2 -25434.808} C_VEL
LIN {X 0,Y 121.942,Z 380.296,A -85,B 0,C 180,E1 -25439.827,E2 -25439.827} C_VEL
LIN {X 0,Y 121.984,Z 380.29,A -85,B 0,C 180,E1 -25446.216,E2 -25446.216} C_VEL
LIN {X 0,Y 122.05,Z 380.278,A -85,B 0,C 180,E1 -25449.788,E2 -25449.788} C_VEL
LIN {X 0,Y 122.265,Z 380.254,A -85,B 0,C 180,E1 -25456.708,E2 -25456.708} C_VEL
LIN {X 0,Y 122.458,Z 380.225,A -85,B 0,C 180,E1 -25460.086,E2 -25460.086} C_VEL
LIN {X 0,Y 122.614,Z 380.208,A -85,B 0,C 180,E1 -25466.714,E2 -25466.714} C_VEL
LIN {X 0,Y 123.046,Z 380.158,A -85,B 0,C 180,E1 -25470,E2 -25470} C_VEL
LIN {X 0,Y 122.446,Z 380.227,A -85,B 0,C 180,E1 -25476.592,E2 -25476.592} C_VEL
LIN {X 0,Y 122.446,Z 380.232,A -85,B 0,C 180,E1 -25479.915,E2 -25479.915} C_VEL
LIN {X 0,Y 122.263,Z 380.251,A -85,B 0,C 180,E1 -25483.293,E2 -25483.293} C_VEL
LIN {X 0,Y 122.055,Z 380.28,A -85,B 0,C 180,E1 -25490.211,E2 -25490.211} C_VEL
LIN {X 0,Y 122.01,Z 380.457,A -85,B 0,C 180,E1 -25496.398,E2 -25496.398} C_VEL
LIN {X 0,Y 122.323,Z 381.592,A -85,B 0,C 180,E1 -25497.016,E2 -25497.016} C_VEL
LIN {X 0,Y 125.957,Z 393.432,A -85,B 0,C 180,E1 -25500.143,E2 -25500.143} C_VEL
LIN {X 0,Y 128.901,Z 404.542,A -85,B 0,C 180,E1 -25503.424,E2 -25503.424} C_VEL
LIN {X 0,Y 130.182,Z 409.734,A -85,B 0,C 180,E1 -25505.111,E2 -25505.111} C_VEL
LIN {X 0,Y 129.027,Z 416.444,A -85,B 0,C 180,E1 -25507.203,E2 -25507.203} C_VEL
LIN {X 0,Y 126.493,Z 428.057,A -85,B 0,C 180,E1 -25511.523,E2 -25511.523} C_VEL
LIN {X 0,Y 124.501,Z 438.026,A -85,B 0,C 180,E1 -25516.251,E2 -25516.251} C_VEL
LIN {X 0,Y 123.124,Z 446.286,A -85,B 0,C 180,E1 -25521.106,E2 -25521.106} C_VEL
LIN {X 0,Y 122.372,Z 453.004,A -85,B 0,C 180,E1 -25525.947,E2 -25525.947} C_VEL
LIN {X 0,Y 122.352,Z 458.818,A -85,B 0,C 180,E1 -25531.127,E2 -25531.127} C_VEL
LIN {X 0,Y 123.191,Z 463.632,A -85,B 0,C 180,E1 -25536.463,E2 -25536.463} C_VEL
LIN {X 0,Y 125.304,Z 467.787,A -85,B 0,C 180,E1 -25542.452,E2 -25542.452} C_VEL
LIN {X 0,Y 128.974,Z 470.858,A -85,B 0,C 180,E1 -25548.761,E2 -25548.761} C_VEL
LIN {X 0,Y 134.092,Z 472.36,A -85,B 0,C 180,E1 -25554.745,E2 -25554.745} C_VEL
LIN {X 0,Y 140.558,Z 472.371,A -85,B 0,C 180,E1 -25560.309,E2 -25560.309} C_VEL
LIN {X 0,Y 148.219,Z 470.78,A -85,B 0,C 180,E1 -25565.304,E2 -25565.304} C_VEL
LIN {X 0,Y 152.971,Z 469.225,A -85,B 0,C 180,E1 -25567.922,E2 -25567.922} C_VEL
LIN {X 0,Y 160.323,Z 465.998,A -85,B 0,C 180,E1 -25571.377,E2 -25571.377} C_VEL
LIN {X 0,Y 166.59,Z 462.578,A -85,B 0,C 180,E1 -25574.003,E2 -25574.003} C_VEL
LIN {X 0,Y 167.411,Z 462.069,A -85,B 0,C 180,E1 -25574.589,E2 -25574.589} C_VEL
LIN {X 0,Y 169.169,Z 460.772,A -85,B 0,C 180,E1 -25577.158,E2 -25577.158} C_VEL
LIN {X 0,Y 169.802,Z 460.273,A -85,B 0,C 180,E1 -25579.337,E2 -25579.337} C_VEL
LIN {X 0,Y 169.907,Z 460.347,A -85,B 0,C 180,E1 -25581.856,E2 -25581.856} C_VEL
LIN {X 0,Y 169.625,Z 460.952,A -85,B 0,C 180,E1 -25584.477,E2 -25584.477} C_VEL
LIN {X 0,Y 169.245,Z 461.95,A -85,B 0,C 180,E1 -25587.18,E2 -25587.18} C_VEL
LIN {X 0,Y 168.742,Z 463.501,A -85,B 0,C 180,E1 -25589.986,E2 -25589.986} C_VEL
LIN {X 0,Y 168.191,Z 465.761,A -85,B 0,C 180,E1 -25593.312,E2 -25593.312} C_VEL
LIN {X 0,Y 167.476,Z 467.456,A -85,B 0,C 180,E1 -25595.087,E2 -25595.087} C_VEL
LIN {X 0,Y 163.057,Z 472.071,A -85,B 0,C 180,E1 -25597.807,E2 -25597.807} C_VEL
LIN {X 0,Y 157.805,Z 477.079,A -85,B 0,C 180,E1 -25600.791,E2 -25600.791} C_VEL
LIN {X 0,Y 151.773,Z 482.169,A -85,B 0,C 180,E1 -25604.145,E2 -25604.145} C_VEL
LIN {X 0,Y 143.741,Z 487.856,A -85,B 0,C 180,E1 -25608.697,E2 -25608.697} C_VEL
LIN {X 0,Y 138.156,Z 491.283,A -85,B 0,C 180,E1 -25612.38,E2 -25612.38} C_VEL
LIN {X 0,Y 131.478,Z 494.684,A -85,B 0,C 180,E1 -25617.688,E2 -25617.688} C_VEL
LIN {X 0,Y 126.201,Z 496.829,A -85,B 0,C 180,E1 -25623.545,E2 -25623.545} C_VEL
LIN {X 0,Y 122.948,Z 497.796,A -85,B 0,C 180,E1 -25629.942,E2 -25629.942} C_VEL
LIN {X 0,Y 121.548,Z 497.547,A -85,B 0,C 180,E1 -25636.628,E2 -25636.628} C_VEL
LIN {X 0,Y 122.019,Z 495.966,A -85,B 0,C 180,E1 -25643.385,E2 -25643.385} C_VEL
LIN {X 0,Y 122.885,Z 494.661,A -85,B 0,C 180,E1 -25646.721,E2 -25646.721} C_VEL
LIN {X 0,Y 123.694,Z 492.864,A -85,B 0,C 180,E1 -25650,E2 -25650} C_VEL
LIN {X 0,Y 122.706,Z 488.449,A -85,B 0,C 180,E1 -25654.928,E2 -25654.928} C_VEL
LIN {X 0,Y 122.379,Z 482.726,A -85,B 0,C 180,E1 -25659.92,E2 -25659.92} C_VEL
LIN {X 0,Y 122.766,Z 475.464,A -85,B 0,C 180,E1 -25664.928,E2 -25664.928} C_VEL
LIN {X 0,Y 123.876,Z 468.095,A -85,B 0,C 180,E1 -25669.039,E2 -25669.039} C_VEL
LIN {X 0,Y 123.881,Z 460.44,A -85,B 0,C 180,E1 -25672.515,E2 -25672.515} C_VEL
LIN {X 0,Y 123.937,Z 450.268,A -85,B 0,C 180,E1 -25676.363,E2 -25676.363} C_VEL
LIN {X 0,Y 124.165,Z 438.005,A -85,B 0,C 180,E1 -25680.154,E2 -25680.154} C_VEL
LIN {X 0,Y 124.276,Z 424.855,A -85,B 0,C 180,E1 -25683.36,E2 -25683.36} C_VEL
LIN {X 0,Y 124.38,Z 411.489,A -85,B 0,C 180,E1 -25685.889,E2 -25685.889} C_VEL
LIN {X 0,Y 124.426,Z 395.988,A -85,B 0,C 180,E1 -25688.129,E2 -25688.129} C_VEL
LIN {X 0,Y 125.07,Z 393.699,A -85,B 0,C 180,E1 -25690.255,E2 -25690.255} C_VEL
LIN {X 0,Y 124.612,Z 391.342,A -85,B 0,C 180,E1 -25692.845,E2 -25692.845} C_VEL
LIN {X 0,Y 123.207,Z 385.581,A -85,B 0,C 180,E1 -25699.378,E2 -25699.378} C_VEL
LIN {X 0,Y 122.16,Z 380.336,A -85,B 0,C 180,E1 -25705.755,E2 -25705.755} C_VEL
LIN {X 0,Y 121.954,Z 380.292,A -85,B 0,C 180,E1 -25712.546,E2 -25712.546} C_VEL
LIN {X 0,Y 122.019,Z 380.278,A -85,B 0,C 180,E1 -25717.152,E2 -25717.152} C_VEL
LIN {X 0,Y 122.072,Z 380.277,A -85,B 0,C 180,E1 -25723.27,E2 -25723.27} C_VEL
LIN {X 0,Y 122.37,Z 380.236,A -85,B 0,C 180,E1 -25729.814,E2 -25729.814} C_VEL
LIN {X 0,Y 121.883,Z 380.311,A -85,B 0,C 180,E1 -25732.569,E2 -25732.569} C_VEL
LIN {X 0,Y 120.414,Z 380.499,A -85,B 0,C 180,E1 -25735.294,E2 -25735.294} C_VEL
LIN {X 0,Y 115.822,Z 381.056,A -85,B 0,C 180,E1 -25742.835,E2 -25742.835} C_VEL
LIN {X 0,Y 115.418,Z 381.099,A -85,B 0,C 180,E1 -25744.838,E2 -25744.838} C_VEL
LIN {X 0,Y 115.36,Z 381.115,A -85,B 0,C 180,E1 -25750.531,E2 -25750.531} C_VEL
LIN {X 0,Y 115.143,Z 381.136,A -85,B 0,C 180,E1 -25754.131,E2 -25754.131} C_VEL
LIN {X 0,Y 114.978,Z 381.156,A -85,B 0,C 180,E1 -25761.515,E2 -25761.515} C_VEL
LIN {X 0,Y 114.869,Z 381.176,A -85,B 0,C 180,E1 -25765.358,E2 -25765.358} C_VEL
LIN {X 0,Y 114.867,Z 381.173,A -85,B 0,C 180,E1 -25771.069,E2 -25771.069} C_VEL
LIN {X 0,Y 114.81,Z 381.178,A -85,B 0,C 180,E1 -25777.745,E2 -25777.745} C_VEL
LIN {X 0,Y 114.807,Z 381.184,A -85,B 0,C 180,E1 -25782.729,E2 -25782.729} C_VEL
LIN {X 0,Y 114.803,Z 381.18,A -85,B 0,C 180,E1 -25787.672,E2 -25787.672} C_VEL
LIN {X 0,Y 114.812,Z 381.181,A -85,B 0,C 180,E1 -25792.728,E2 -25792.728} C_VEL
LIN {X 0,Y 114.869,Z 381.176,A -85,B 0,C 180,E1 -25798.933,E2 -25798.933} C_VEL
LIN {X 0,Y 114.947,Z 381.166,A -85,B 0,C 180,E1 -25806.508,E2 -25806.508} C_VEL
LIN {X 0,Y 115.019,Z 381.153,A -85,B 0,C 180,E1 -25812.211,E2 -25812.211} C_VEL
LIN {X 0,Y 115.287,Z 381.124,A -85,B 0,C 180,E1 -25817.258,E2 -25817.258} C_VEL
LIN {X 0,Y 115.395,Z 381.104,A -85,B 0,C 180,E1 -25819.472,E2 -25819.472} C_VEL
LIN {X 0,Y 115.54,Z 381.089,A -85,B 0,C 180,E1 -25826.513,E2 -25826.513} C_VEL
LIN {X 0,Y 115.997,Z 381.036,A -85,B 0,C 180,E1 -25830,E2 -25830} C_VEL
LIN {X 0,Y 115.388,Z 381.107,A -85,B 0,C 180,E1 -25836.997,E2 -25836.997} C_VEL
LIN {X 0,Y 115.285,Z 381.118,A -85,B 0,C 180,E1 -25842.737,E2 -25842.737} C_VEL
LIN {X 0,Y 115.017,Z 381.155,A -85,B 0,C 180,E1 -25847.789,E2 -25847.789} C_VEL
LIN {X 0,Y 114.935,Z 381.167,A -85,B 0,C 180,E1 -25854.231,E2 -25854.231} C_VEL
LIN {X 0,Y 114.962,Z 381.361,A -85,B 0,C 180,E1 -25855.336,E2 -25855.336} C_VEL
LIN {X 0,Y 115.271,Z 382.559,A -85,B 0,C 180,E1 -25855.99,E2 -25855.99} C_VEL
LIN {X 0,Y 118.833,Z 394.011,A -85,B 0,C 180,E1 -25859.203,E2 -25859.203} C_VEL
LIN {X 0,Y 121.833,Z 405.257,A -85,B 0,C 180,E1 -25862.737,E2 -25862.737} C_VEL
LIN {X 0,Y 123.204,Z 411.218,A -85,B 0,C 180,E1 -25864.78,E2 -25864.78} C_VEL
LIN {X 0,Y 120.817,Z 422.121,A -85,B 0,C 180,E1 -25868.52,E2 -25868.52} C_VEL
LIN {X 0,Y 118.406,Z 433.296,A -85,B 0,C 180,E1 -25873.356,E2 -25873.356} C_VEL
LIN {X 0,Y 116.627,Z 442.592,A -85,B 0,C 180,E1 -25878.481,E2 -25878.481} C_VEL
LIN {X 0,Y 115.549,Z 450.121,A -85,B 0,C 180,E1 -25883.628,E2 -25883.628} C_VEL
LIN {X 0,Y 115.183,Z 457.371,A -85,B 0,C 180,E1 -25889.747,E2 -25889.747} C_VEL
LIN {X 0,Y 115.862,Z 462.78,A -85,B 0,C 180,E1 -25895.484,E2 -25895.484} C_VEL
LIN {X 0,Y 118.013,Z 467.792,A -85,B 0,C 180,E1 -25902.329,E2 -25902.329} C_VEL
LIN {X 0,Y 121.72,Z 471.291,A -85,B 0,C 180,E1 -25908.973,E2 -25908.973} C_VEL
LIN {X 0,Y 126.941,Z 473.282,A -85,B 0,C 180,E1 -25915.228,E2 -25915.228} C_VEL
LIN {X 0,Y 133.549,Z 473.79,A -85,B 0,C 180,E1 -25921.013,E2 -25921.013} C_VEL
LIN {X 0,Y 141.376,Z 472.745,A -85,B 0,C 180,E1 -25926.171,E2 -25926.171} C_VEL
LIN {X 0,Y 150.251,Z 470.176,A -85,B 0,C 180,E1 -25930.811,E2 -25930.811} C_VEL
LIN {X 0,Y 159.962,Z 465.96,A -85,B 0,C 180,E1 -25934.86,E2 -25934.86} C_VEL
LIN {X 0,Y 160.822,Z 465.538,A -85,B 0,C 180,E1 -25935.201,E2 -25935.201} C_VEL
LIN {X 0,Y 163.112,Z 464.269,A -85,B 0,C 180,E1 -25937.554,E2 -25937.554} C_VEL
LIN {X 0,Y 163.765,Z 464.011,A -85,B 0,C 180,E1 -25940.079,E2 -25940.079} C_VEL
LIN {X 0,Y 163.766,Z 464.334,A -85,B 0,C 180,E1 -25942.721,E2 -25942.721} C_VEL
LIN {X 0,Y 163.464,Z 465.193,A -85,B 0,C 180,E1 -25945.464,E2 -25945.464} C_VEL
LIN {X 0,Y 162.612,Z 467.525,A -85,B 0,C 180,E1 -25950.19,E2 -25950.19} C_VEL
LIN {X 0,Y 162.188,Z 469.045,A -85,B 0,C 180,E1 -25952.634,E2 -25952.634} C_VEL
LIN {X 0,Y 161.358,Z 470.443,A -85,B 0,C 180,E1 -25954.154,E2 -25954.154} C_VEL
LIN {X 0,Y 157.317,Z 474.103,A -85,B 0,C 180,E1 -25956.475,E2 -25956.475} C_VEL
LIN {X 0,Y 151.071,Z 479.253,A -85,B 0,C 180,E1 -25959.863,E2 -25959.863} C_VEL
LIN {X 0,Y 144.739,Z 483.787,A -85,B 0,C 180,E1 -25963.254,E2 -25963.254} C_VEL
LIN {X 0,Y 136.409,Z 488.797,A -85,B 0,C 180,E1 -25967.951,E2 -25967.951} C_VEL
LIN {X 0,Y 128.878,Z 492.54,A -85,B 0,C 180,E1 -25973.142,E2 -25973.142} C_VEL
LIN {X 0,Y 122.494,Z 495.043,A -85,B 0,C 180,E1 -25978.912,E2 -25978.912} C_VEL
LIN {X 0,Y 117.861,Z 496.315,A -85,B 0,C 180,E1 -25985.33,E2 -25985.33} C_VEL
LIN {X 0,Y 115.25,Z 496.399,A -85,B 0,C 180,E1 -25992.248,E2 -25992.248} C_VEL
LIN {X 0,Y 114.66,Z 495.289,A -85,B 0,C 180,E1 -25999.404,E2 -25999.404} C_VEL
LIN {X 0,Y 115.973,Z 492.825,A -85,B 0,C 180,E1 -26006.526,E2 -26006.526} C_VEL
LIN {X 0,Y 116.731,Z 490.894,A -85,B 0,C 180,E1 -26010,E2 -26010} C_VEL
LIN {X 0,Y 115.704,Z 486.234,A -85,B 0,C 180,E1 -26015.227,E2 -26015.227} C_VEL
LIN {X 0,Y 115.45,Z 480.236,A -85,B 0,C 180,E1 -26020.522,E2 -26020.522} C_VEL
LIN {X 0,Y 115.973,Z 472.653,A -85,B 0,C 180,E1 -26025.825,E2 -26025.825} C_VEL
LIN {X 0,Y 116.893,Z 466.587,A -85,B 0,C 180,E1 -26029.309,E2 -26029.309} C_VEL
LIN {X 0,Y 116.833,Z 457.7,A -85,B 0,C 180,E1 -26033.485,E2 -26033.485} C_VEL
LIN {X 0,Y 116.959,Z 446.451,A -85,B 0,C 180,E1 -26037.84,E2 -26037.84} C_VEL
LIN {X 0,Y 117.176,Z 434.146,A -85,B 0,C 180,E1 -26041.655,E2 -26041.655} C_VEL
LIN {X 0,Y 117.38,Z 422.061,A -85,B 0,C 180,E1 -26044.664,E2 -26044.664} C_VEL
LIN {X 0,Y 117.509,Z 408.124,A -85,B 0,C 180,E1 -26047.316,E2 -26047.316} C_VEL
LIN {X 0,Y 117.625,Z 395.03,A -85,B 0,C 180,E1 -26049.254,E2 -26049.254} C_VEL
LIN {X 0,Y 117.871,Z 393.222,A -85,B 0,C 180,E1 -26050.985,E2 -26050.985} C_VEL
LIN {X 0,Y 116.735,Z 388.773,A -85,B 0,C 180,E1 -26056.256,E2 -26056.256} C_VEL
LIN {X 0,Y 115.589,Z 383.657,A -85,B 0,C 180,E1 -26062.553,E2 -26062.553} C_VEL
LIN {X 0,Y 115.094,Z 381.207,A -85,B 0,C 180,E1 -26065.874,E2 -26065.874} C_VEL
LIN {X 0,Y 114.893,Z 381.169,A -85,B 0,C 180,E1 -26070.701,E2 -26070.701} C_VEL
LIN {X 0,Y 114.942,Z 381.162,A -85,B 0,C 180,E1 -26076.51,E2 -26076.51} C_VEL
LIN {X 0,Y 114.981,Z 381.162,A -85,B 0,C 180,E1 -26082.205,E2 -26082.205} C_VEL
LIN {X 0,Y 115.306,Z 381.116,A -85,B 0,C 180,E1 -26089.464,E2 -26089.464} C_VEL
LIN {X 0,Y 115.513,Z 381.09,A -85,B 0,C 180,E1 -26096.512,E2 -26096.512} C_VEL
LIN {X 0,Y 115.988,Z 381.036,A -85,B 0,C 180,E1 -26100,E2 -26100} C_VEL
LIN {X 0,Y 115.418,Z 381.099,A -85,B 0,C 180,E1 -26104.838,E2 -26104.838} C_VEL
LIN {X 0,Y 114.604,Z 381.209,A -85,B 0,C 180,E1 -26107.747,E2 -26107.747} C_VEL
LIN {X 0,Y 112.907,Z 381.42,A -85,B 0,C 180,E1 -26110.618,E2 -26110.618} C_VEL
LIN {X 0,Y 108.172,Z 382.01,A -85,B 0,C 180,E1 -26118.612,E2 -26118.612} C_VEL
LIN {X 0,Y 107.841,Z 382.041,A -85,B 0,C 180,E1 -26120.745,E2 -26120.745} C_VEL
LIN {X 0,Y 107.856,Z 382.048,A -85,B 0,C 180,E1 -26124.184,E2 -26124.184} C_VEL
LIN {X 0,Y 107.793,Z 382.055,A -85,B 0,C 180,E1 -26132.052,E2 -26132.052} C_VEL
LIN {X 0,Y 107.715,Z 382.061,A -85,B 0,C 180,E1 -26138.47,E2 -26138.47} C_VEL
LIN {X 0,Y 107.687,Z 382.065,A -85,B 0,C 180,E1 -26145.881,E2 -26145.881} C_VEL
LIN {X 0,Y 107.708,Z 382.068,A -85,B 0,C 180,E1 -26151.537,E2 -26151.537} C_VEL
LIN {X 0,Y 107.807,Z 382.056,A -85,B 0,C 180,E1 -26158.566,E2 -26158.566} C_VEL
LIN {X 0,Y 107.911,Z 382.043,A -85,B 0,C 180,E1 -26166.999,E2 -26166.999} C_VEL
LIN {X 0,Y 108.041,Z 382.026,A -85,B 0,C 180,E1 -26174.919,E2 -26174.919} C_VEL
LIN {X 0,Y 108.308,Z 381.988,A -85,B 0,C 180,E1 -26178.775,E2 -26178.775} C_VEL
LIN {X 0,Y 108.466,Z 381.97,A -85,B 0,C 180,E1 -26186.285,E2 -26186.285} C_VEL
LIN {X 0,Y 108.947,Z 381.915,A -85,B 0,C 180,E1 -26190,E2 -26190} C_VEL
LIN {X 0,Y 108.328,Z 381.988,A -85,B 0,C 180,E1 -26197.455,E2 -26197.455} C_VEL
LIN {X 0,Y 108.2,Z 382.001,A -85,B 0,C 180,E1 -26203.015,E2 -26203.015} C_VEL
LIN {X 0,Y 107.91,Z 382.045,A -85,B 0,C 180,E1 -26209.004,E2 -26209.004} C_VEL
LIN {X 0,Y 107.917,Z 382.236,A -85,B 0,C 180,E1 -26214.177,E2 -26214.177} C_VEL
LIN {X 0,Y 108.131,Z 383.169,A -85,B 0,C 180,E1 -26214.789,E2 -26214.789} C_VEL
LIN {X 0,Y 111.995,Z 395.608,A -85,B 0,C 180,E1 -26218.533,E2 -26218.533} C_VEL
LIN {X 0,Y 115.002,Z 406.977,A -85,B 0,C 180,E1 -26222.325,E2 -26222.325} C_VEL
LIN {X 0,Y 116.075,Z 411.73,A -85,B 0,C 180,E1 -26224.059,E2 -26224.059} C_VEL
LIN {X 0,Y 114.365,Z 419.997,A -85,B 0,C 180,E1 -26226.976,E2 -26226.976} C_VEL
LIN {X 0,Y 112.108,Z 429.94,A -85,B 0,C 180,E1 -26231.212,E2 -26231.212} C_VEL
LIN {X 0,Y 109.999,Z 440.03,A -85,B 0,C 180,E1 -26236.62,E2 -26236.62} C_VEL
LIN {X 0,Y 108.623,Z 448.794,A -85,B 0,C 180,E1 -26242.503,E2 -26242.503} C_VEL
LIN {X 0,Y 108.059,Z 456.128,A -85,B 0,C 180,E1 -26248.647,E2 -26248.647} C_VEL
LIN {X 0,Y 108.626,Z 462.131,A -85,B 0,C 180,E1 -26254.927,E2 -26254.927} C_VEL
LIN {X 0,Y 110.718,Z 467.639,A -85,B 0,C 180,E1 -26262.198,E2 -26262.198} C_VEL
LIN {X 0,Y 114.463,Z 471.577,A -85,B 0,C 180,E1 -26269.225,E2 -26269.225} C_VEL
LIN {X 0,Y 119.793,Z 474.063,A -85,B 0,C 180,E1 -26275.808,E2 -26275.808} C_VEL
LIN {X 0,Y 126.565,Z 475.035,A -85,B 0,C 180,E1 -26281.83,E2 -26281.83} C_VEL
LIN {X 0,Y 134.571,Z 474.535,A -85,B 0,C 180,E1 -26287.137,E2 -26287.137} C_VEL
LIN {X 0,Y 143.629,Z 472.554,A -85,B 0,C 180,E1 -26291.872,E2 -26291.872} C_VEL
LIN {X 0,Y 153.51,Z 469,A -85,B 0,C 180,E1 -26295.972,E2 -26295.972} C_VEL
LIN {X 0,Y 157.026,Z 467.517,A -85,B 0,C 180,E1 -26298.258,E2 -26298.258} C_VEL
LIN {X 0,Y 157.525,Z 467.552,A -85,B 0,C 180,E1 -26300.911,E2 -26300.911} C_VEL
LIN {X 0,Y 157.429,Z 468.148,A -85,B 0,C 180,E1 -26303.69,E2 -26303.69} C_VEL
LIN {X 0,Y 156.984,Z 469.222,A -85,B 0,C 180,E1 -26306.596,E2 -26306.596} C_VEL
LIN {X 0,Y 156.113,Z 471.617,A -85,B 0,C 180,E1 -26311.203,E2 -26311.203} C_VEL
LIN {X 0,Y 155.494,Z 472.775,A -85,B 0,C 180,E1 -26312.846,E2 -26312.846} C_VEL
LIN {X 0,Y 153.064,Z 474.801,A -85,B 0,C 180,E1 -26314.264,E2 -26314.264} C_VEL
LIN {X 0,Y 146.512,Z 479.56,A -85,B 0,C 180,E1 -26317.677,E2 -26317.677} C_VEL
LIN {X 0,Y 139.912,Z 483.849,A -85,B 0,C 180,E1 -26321.11,E2 -26321.11} C_VEL
LIN {X 0,Y 131.194,Z 488.463,A -85,B 0,C 180,E1 -26325.862,E2 -26325.862} C_VEL
LIN {X 0,Y 123.253,Z 491.878,A -85,B 0,C 180,E1 -26331.155,E2 -26331.155} C_VEL
LIN {X 0,Y 116.464,Z 494.064,A -85,B 0,C 180,E1 -26337.106,E2 -26337.106} C_VEL
LIN {X 0,Y 111.437,Z 495.073,A -85,B 0,C 180,E1 -26343.803,E2 -26343.803} C_VEL
LIN {X 0,Y 108.536,Z 494.95,A -85,B 0,C 180,E1 -26351.11,E2 -26351.11} C_VEL
LIN {X 0,Y 107.808,Z 493.607,A -85,B 0,C 180,E1 -26358.722,E2 -26358.722} C_VEL
LIN {X 0,Y 109.068,Z 490.919,A -85,B 0,C 180,E1 -26366.306,E2 -26366.306} C_VEL
LIN {X 0,Y 109.772,Z 488.811,A -85,B 0,C 180,E1 -26370,E2 -26370} C_VEL
LIN {X 0,Y 108.741,Z 483.882,A -85,B 0,C 180,E1 -26375.563,E2 -26375.563} C_VEL
LIN {X 0,Y 108.539,Z 477.588,A -85,B 0,C 180,E1 -26381.201,E2 -26381.201} C_VEL
LIN {X 0,Y 109.248,Z 469.657,A -85,B 0,C 180,E1 -26386.827,E2 -26386.827} C_VEL
LIN {X 0,Y 109.863,Z 464.918,A -85,B 0,C 180,E1 -26389.623,E2 -26389.623} C_VEL
LIN {X 0,Y 109.736,Z 454.744,A -85,B 0,C 180,E1 -26394.6,E2 -26394.6} C_VEL
LIN {X 0,Y 109.894,Z 444.556,A -85,B 0,C 180,E1 -26398.661,E2 -26398.661} C_VEL
LIN {X 0,Y 110.138,Z 433.524,A -85,B 0,C 180,E1 -26402.283,E2 -26402.283} C_VEL
LIN {X 0,Y 110.434,Z 421.438,A -85,B 0,C 180,E1 -26405.5,E2 -26405.5} C_VEL
LIN {X 0,Y 110.654,Z 407.98,A -85,B 0,C 180,E1 -26408.261,E2 -26408.261} C_VEL
LIN {X 0,Y 110.743,Z 394.108,A -85,B 0,C 180,E1 -26410.512,E2 -26410.512} C_VEL
LIN {X 0,Y 110.637,Z 392.816,A -85,B 0,C 180,E1 -26411.632,E2 -26411.632} C_VEL
LIN {X 0,Y 109.385,Z 388.138,A -85,B 0,C 180,E1 -26417.574,E2 -26417.574} C_VEL
LIN {X 0,Y 108.14,Z 382.361,A -85,B 0,C 180,E1 -26425.242,E2 -26425.242} C_VEL
LIN {X 0,Y 108.018,Z 382.043,A -85,B 0,C 180,E1 -26426.224,E2 -26426.224} C_VEL
LIN {X 0,Y 107.855,Z 382.047,A -85,B 0,C 180,E1 -26435.817,E2 -26435.817} C_VEL
LIN {X 0,Y 107.881,Z 382.047,A -85,B 0,C 180,E1 -26440.99,E2 -26440.99} C_VEL
LIN {X 0,Y 108.223,Z 381.995,A -85,B 0,C 180,E1 -26448.766,E2 -26448.766} C_VEL
LIN {X 0,Y 108.436,Z 381.972,A -85,B 0,C 180,E1 -26456.284,E2 -26456.284} C_VEL
LIN {X 0,Y 108.913,Z 381.917,A -85,B 0,C 180,E1 -26460,E2 -26460} C_VEL
LIN {X 0,Y 108.322,Z 381.99,A -85,B 0,C 180,E1 -26467.456,E2 -26467.456} C_VEL
LIN {X 0,Y 108.196,Z 382,A -85,B 0,C 180,E1 -26473.014,E2 -26473.014} C_VEL
LIN {X 0,Y 107.841,Z 382.041,A -85,B 0,C 180,E1 -26480.745,E2 -26480.745} C_VEL
LIN {X 0,Y 107.123,Z 382.14,A -85,B 0,C 180,E1 -26483.858,E2 -26483.858} C_VEL
LIN {X 0,Y 105.47,Z 382.346,A -85,B 0,C 180,E1 -26486.933,E2 -26486.933} C_VEL
LIN {X 0,Y 100.842,Z 382.923,A -85,B 0,C 180,E1 -26495.532,E2 -26495.532} C_VEL
LIN {X 0,Y 100.593,Z 382.942,A -85,B 0,C 180,E1 -26497.826,E2 -26497.826} C_VEL
LIN {X 0,Y 100.66,Z 382.944,A -85,B 0,C 180,E1 -26504.282,E2 -26504.282} C_VEL
LIN {X 0,Y 100.645,Z 382.948,A -85,B 0,C 180,E1 -26511.064,E2 -26511.064} C_VEL
LIN {X 0,Y 100.7,Z 382.939,A -85,B 0,C 180,E1 -26516.877,E2 -26516.877} C_VEL
LIN {X 0,Y 100.786,Z 382.928,A -85,B 0,C 180,E1 -26525.268,E2 -26525.268} C_VEL
LIN {X 0,Y 100.819,Z 382.923,A -85,B 0,C 180,E1 -26529.602,E2 -26529.602} C_VEL
LIN {X 0,Y 101.2,Z 382.875,A -85,B 0,C 180,E1 -26537.975,E2 -26537.975} C_VEL
LIN {X 0,Y 101.281,Z 382.868,A -85,B 0,C 180,E1 -26542.023,E2 -26542.023} C_VEL
LIN {X 0,Y 101.871,Z 382.796,A -85,B 0,C 180,E1 -26550,E2 -26550} C_VEL
LIN {X 0,Y 101.267,Z 382.87,A -85,B 0,C 180,E1 -26557.978,E2 -26557.978} C_VEL
LIN {X 0,Y 101.125,Z 382.883,A -85,B 0,C 180,E1 -26563.351,E2 -26563.351} C_VEL
LIN {X 0,Y 100.871,Z 383.06,A -85,B 0,C 180,E1 -26572.802,E2 -26572.802} C_VEL
LIN {X 0,Y 101.134,Z 384.128,A -85,B 0,C 180,E1 -26573.551,E2 -26573.551} C_VEL
LIN {X 0,Y 104.691,Z 395.551,A -85,B 0,C 180,E1 -26577.248,E2 -26577.248} C_VEL
LIN {X 0,Y 107.493,Z 406.126,A -85,B 0,C 180,E1 -26580.988,E2 -26580.988} C_VEL
LIN {X 0,Y 109.088,Z 412.905,A -85,B 0,C 180,E1 -26583.601,E2 -26583.601} C_VEL
LIN {X 0,Y 106.562,Z 423.553,A -85,B 0,C 180,E1 -26587.681,E2 -26587.681} C_VEL
LIN {X 0,Y 104.23,Z 433.752,A -85,B 0,C 180,E1 -26592.613,E2 -26592.613} C_VEL
LIN {X 0,Y 102.415,Z 442.954,A -85,B 0,C 180,E1 -26598.15,E2 -26598.15} C_VEL
LIN {X 0,Y 101.32,Z 450.633,A -85,B 0,C 180,E1 -26603.872,E2 -26603.872} C_VEL
LIN {X 0,Y 101.049,Z 458.15,A -85,B 0,C 180,E1 -26610.866,E2 -26610.866} C_VEL
LIN {X 0,Y 102.097,Z 464.153,A -85,B 0,C 180,E1 -26617.753,E2 -26617.753} C_VEL
LIN {X 0,Y 104.391,Z 468.826,A -85,B 0,C 180,E1 -26624.378,E2 -26624.378} C_VEL
LIN {X 0,Y 107.204,Z 471.706,A -85,B 0,C 180,E1 -26629.526,E2 -26629.526} C_VEL
LIN {X 0,Y 112.66,Z 474.659,A -85,B 0,C 180,E1 -26636.464,E2 -26636.464} C_VEL
LIN {X 0,Y 119.61,Z 476.12,A -85,B 0,C 180,E1 -26642.744,E2 -26642.744} C_VEL
LIN {X 0,Y 127.822,Z 476.165,A -85,B 0,C 180,E1 -26648.247,E2 -26648.247} C_VEL
LIN {X 0,Y 137.074,Z 474.716,A -85,B 0,C 180,E1 -26653.06,E2 -26653.06} C_VEL
LIN {X 0,Y 147.143,Z 471.839,A -85,B 0,C 180,E1 -26657.208,E2 -26657.208} C_VEL
LIN {X 0,Y 150.675,Z 470.601,A -85,B 0,C 180,E1 -26659.057,E2 -26659.057} C_VEL
LIN {X 0,Y 151.084,Z 470.894,A -85,B 0,C 180,E1 -26661.848,E2 -26661.848} C_VEL
LIN {X 0,Y 150.851,Z 471.746,A -85,B 0,C 180,E1 -26664.791,E2 -26664.791} C_VEL
LIN {X 0,Y 150.282,Z 473.035,A -85,B 0,C 180,E1 -26667.882,E2 -26667.882} C_VEL
LIN {X 0,Y 149.579,Z 474.734,A -85,B 0,C 180,E1 -26671.121,E2 -26671.121} C_VEL
LIN {X 0,Y 149.02,Z 475.355,A -85,B 0,C 180,E1 -26671.909,E2 -26671.909} C_VEL
LIN {X 0,Y 142.181,Z 479.852,A -85,B 0,C 180,E1 -26675.356,E2 -26675.356} C_VEL
LIN {X 0,Y 135.278,Z 483.771,A -85,B 0,C 180,E1 -26678.806,E2 -26678.806} C_VEL
LIN {X 0,Y 126.149,Z 488.074,A -85,B 0,C 180,E1 -26683.595,E2 -26683.595} C_VEL
LIN {X 0,Y 117.794,Z 491.177,A -85,B 0,C 180,E1 -26688.983,E2 -26688.983} C_VEL
LIN {X 0,Y 110.576,Z 493.071,A -85,B 0,C 180,E1 -26695.11,E2 -26695.11} C_VEL
LIN {X 0,Y 105.113,Z 493.788,A -85,B 0,C 180,E1 -26702.094,E2 -26702.094} C_VEL
LIN {X 0,Y 101.912,Z 493.39,A -85,B 0,C 180,E1 -26709.83,E2 -26709.83} C_VEL
LIN {X 0,Y 100.966,Z 491.815,A -85,B 0,C 180,E1 -26717.947,E2 -26717.947} C_VEL
LIN {X 0,Y 102.206,Z 488.917,A -85,B 0,C 180,E1 -26726.057,E2 -26726.057} C_VEL
LIN {X 0,Y 102.66,Z 487.909,A -85,B 0,C 180,E1 -26728.038,E2 -26728.038} C_VEL
LIN {X 0,Y 102.804,Z 486.7,A -85,B 0,C 180,E1 -26730,E2 -26730} C_VEL
LIN {X 0,Y 101.73,Z 480.494,A -85,B 0,C 180,E1 -26736.944,E2 -26736.944} C_VEL
LIN {X 0,Y 101.711,Z 473.622,A -85,B 0,C 180,E1 -26742.943,E2 -26742.943} C_VEL
LIN {X 0,Y 102.569,Z 466.542,A -85,B 0,C 180,E1 -26747.959,E2 -26747.959} C_VEL
LIN {X 0,Y 102.78,Z 463.16,A -85,B 0,C 180,E1 -26749.992,E2 -26749.992} C_VEL
LIN {X 0,Y 102.665,Z 453.12,A -85,B 0,C 180,E1 -26755.167,E2 -26755.167} C_VEL
LIN {X 0,Y 102.845,Z 442.326,A -85,B 0,C 180,E1 -26759.698,E2 -26759.698} C_VEL
LIN {X 0,Y 103.205,Z 430.218,A -85,B 0,C 180,E1 -26763.836,E2 -26763.836} C_VEL
LIN {X 0,Y 103.592,Z 417.373,A -85,B 0,C 180,E1 -26767.281,E2 -26767.281} C_VEL
LIN {X 0,Y 103.905,Z 404.38,A -85,B 0,C 180,E1 -26769.983,E2 -26769.983} C_VEL
LIN {X 0,Y 103.97,Z 395.448,A -85,B 0,C 180,E1 -26771.418,E2 -26771.418} C_VEL
LIN {X 0,Y 103.426,Z 392.675,A -85,B 0,C 180,E1 -26772.176,E2 -26772.176} C_VEL
LIN {X 0,Y 101.985,Z 387.324,A -85,B 0,C 180,E1 -26779.289,E2 -26779.289} C_VEL
LIN {X 0,Y 101.01,Z 382.967,A -85,B 0,C 180,E1 -26785.726,E2 -26785.726} C_VEL
LIN {X 0,Y 100.785,Z 382.929,A -85,B 0,C 180,E1 -26795.266,E2 -26795.266} C_VEL
LIN {X 0,Y 100.8,Z 382.925,A -85,B 0,C 180,E1 -26799.597,E2 -26799.597} C_VEL
LIN {X 0,Y 101.122,Z 382.876,A -85,B 0,C 180,E1 -26807.965,E2 -26807.965} C_VEL
LIN {X 0,Y 101.229,Z 382.875,A -85,B 0,C 180,E1 -26812.018,E2 -26812.018} C_VEL
LIN {X 0,Y 101.841,Z 382.798,A -85,B 0,C 180,E1 -26820,E2 -26820} C_VEL
LIN {X 0,Y 101.261,Z 382.87,A -85,B 0,C 180,E1 -26827.979,E2 -26827.979} C_VEL
LIN {X 0,Y 101.122,Z 382.881,A -85,B 0,C 180,E1 -26833.35,E2 -26833.35} C_VEL
LIN {X 0,Y 100.8,Z 382.922,A -85,B 0,C 180,E1 -26840.602,E2 -26840.602} C_VEL
LIN {X 0,Y 100.773,Z 382.932,A -85,B 0,C 180,E1 -26844.959,E2 -26844.959} C_VEL
LIN {X 0,Y 100.699,Z 382.941,A -85,B 0,C 180,E1 -26853.125,E2 -26853.125} C_VEL
LIN {X 0,Y 100.593,Z 382.942,A -85,B 0,C 180,E1 -26857.826,E2 -26857.826} C_VEL
LIN {X 0,Y 100.351,Z 382.981,A -85,B 0,C 180,E1 -26860.059,E2 -26860.059} C_VEL
LIN {X 0,Y 99.599,Z 383.079,A -85,B 0,C 180,E1 -26862.272,E2 -26862.272} C_VEL
LIN {X 0,Y 97.255,Z 383.373,A -85,B 0,C 180,E1 -26866.69,E2 -26866.69} C_VEL
LIN {X 0,Y 93.943,Z 383.779,A -85,B 0,C 180,E1 -26873.745,E2 -26873.745} C_VEL
LIN {X 0,Y 93.58,Z 383.821,A -85,B 0,C 180,E1 -26876.219,E2 -26876.219} C_VEL
LIN {X 0,Y 93.669,Z 383.812,A -85,B 0,C 180,E1 -26884.205,E2 -26884.205} C_VEL
LIN {X 0,Y 93.695,Z 383.814,A -85,B 0,C 180,E1 -26887.973,E2 -26887.973} C_VEL
LIN {X 0,Y 94.099,Z 383.763,A -85,B 0,C 180,E1 -26897.053,E2 -26897.053} C_VEL
LIN {X 0,Y 94.213,Z 383.746,A -85,B 0,C 180,E1 -26901.42,E2 -26901.42} C_VEL
LIN {X 0,Y 94.797,Z 383.677,A -85,B 0,C 180,E1 -26910,E2 -26910} C_VEL
LIN {X 0,Y 94.2,Z 383.751,A -85,B 0,C 180,E1 -26918.581,E2 -26918.581} C_VEL
LIN {X 0,Y 94.043,Z 383.767,A -85,B 0,C 180,E1 -26923.709,E2 -26923.709} C_VEL
LIN {X 0,Y 93.801,Z 383.992,A -85,B 0,C 180,E1 -26931.423,E2 -26931.423} C_VEL
LIN {X 0,Y 94.089,Z 385.148,A -85,B 0,C 180,E1 -26932.218,E2 -26932.218} C_VEL
LIN {X 0,Y 97.697,Z 396.563,A -85,B 0,C 180,E1 -26936.179,E2 -26936.179} C_VEL
LIN {X 0,Y 100.326,Z 406.47,A -85,B 0,C 180,E1 -26939.941,E2 -26939.941} C_VEL
LIN {X 0,Y 102.016,Z 413.504,A -85,B 0,C 180,E1 -26942.854,E2 -26942.854} C_VEL
LIN {X 0,Y 99.38,Z 424.431,A -85,B 0,C 180,E1 -26947.29,E2 -26947.29} C_VEL
LIN {X 0,Y 97.107,Z 434.063,A -85,B 0,C 180,E1 -26952.244,E2 -26952.244} C_VEL
LIN {X 0,Y 95.219,Z 443.562,A -85,B 0,C 180,E1 -26958.373,E2 -26958.373} C_VEL
LIN {X 0,Y 94.073,Z 452.109,A -85,B 0,C 180,E1 -26965.262,E2 -26965.262} C_VEL
LIN {X 0,Y 94.194,Z 460.275,A -85,B 0,C 180,E1 -26973.55,E2 -26973.55} C_VEL
LIN {X 0,Y 95.585,Z 465.632,A -85,B 0,C 180,E1 -26980.276,E2 -26980.276} C_VEL
LIN {X 0,Y 98.68,Z 470.429,A -85,B 0,C 180,E1 -26987.663,E2 -26987.663} C_VEL
LIN {X 0,Y 101.347,Z 472.767,A -85,B 0,C 180,E1 -26992.028,E2 -26992.028} C_VEL
LIN {X 0,Y 105.538,Z 475.088,A -85,B 0,C 180,E1 -26997.258,E2 -26997.258} C_VEL
LIN {X 0,Y 112.693,Z 477.04,A -85,B 0,C 180,E1 -27003.798,E2 -27003.798} C_VEL
LIN {X 0,Y 121.14,Z 477.592,A -85,B 0,C 180,E1 -27009.515,E2 -27009.515} C_VEL
LIN {X 0,Y 130.612,Z 476.694,A -85,B 0,C 180,E1 -27014.415,E2 -27014.415} C_VEL
LIN {X 0,Y 140.891,Z 474.43,A -85,B 0,C 180,E1 -27018.604,E2 -27018.604} C_VEL
LIN {X 0,Y 144.06,Z 473.496,A -85,B 0,C 180,E1 -27019.968,E2 -27019.968} C_VEL
LIN {X 0,Y 144.442,Z 474.047,A -85,B 0,C 180,E1 -27022.908,E2 -27022.908} C_VEL
LIN {X 0,Y 144.033,Z 475.109,A -85,B 0,C 180,E1 -27026.05,E2 -27026.05} C_VEL
LIN {X 0,Y 143.3,Z 476.634,A -85,B 0,C 180,E1 -27029.37,E2 -27029.37} C_VEL
LIN {X 0,Y 142.291,Z 477.643,A -85,B 0,C 180,E1 -27030.835,E2 -27030.835} C_VEL
LIN {X 0,Y 135.663,Z 481.293,A -85,B 0,C 180,E1 -27034.019,E2 -27034.019} C_VEL
LIN {X 0,Y 128.467,Z 484.773,A -85,B 0,C 180,E1 -27037.512,E2 -27037.512} C_VEL
LIN {X 0,Y 121.324,Z 487.594,A -85,B 0,C 180,E1 -27041.146,E2 -27041.146} C_VEL
LIN {X 0,Y 112.523,Z 490.369,A -85,B 0,C 180,E1 -27046.605,E2 -27046.605} C_VEL
LIN {X 0,Y 104.852,Z 491.966,A -85,B 0,C 180,E1 -27052.898,E2 -27052.898} C_VEL
LIN {X 0,Y 98.917,Z 492.418,A -85,B 0,C 180,E1 -27060.176,E2 -27060.176} C_VEL
LIN {X 0,Y 95.337,Z 491.791,A -85,B 0,C 180,E1 -27068.372,E2 -27068.372} C_VEL
LIN {X 0,Y 94.189,Z 489.994,A -85,B 0,C 180,E1 -27077.065,E2 -27077.065} C_VEL
LIN {X 0,Y 95.364,Z 486.834,A -85,B 0,C 180,E1 -27085.774,E2 -27085.774} C_VEL
LIN {X 0,Y 95.872,Z 485.793,A -85,B 0,C 180,E1 -27087.9,E2 -27087.9} C_VEL
LIN {X 0,Y 95.872,Z 484.407,A -85,B 0,C 180,E1 -27090,E2 -27090} C_VEL
LIN {X 0,Y 94.891,Z 478.938,A -85,B 0,C 180,E1 -27096.378,E2 -27096.378} C_VEL
LIN {X 0,Y 94.78,Z 471.972,A -85,B 0,C 180,E1 -27102.853,E2 -27102.853} C_VEL
LIN {X 0,Y 95.63,Z 464.878,A -85,B 0,C 180,E1 -27108.2,E2 -27108.2} C_VEL
LIN {X 0,Y 95.592,Z 457.412,A -85,B 0,C 180,E1 -27112.704,E2 -27112.704} C_VEL
LIN {X 0,Y 95.706,Z 446.344,A -85,B 0,C 180,E1 -27118.212,E2 -27118.212} C_VEL
LIN {X 0,Y 96.03,Z 435.347,A -85,B 0,C 180,E1 -27122.665,E2 -27122.665} C_VEL
LIN {X 0,Y 96.504,Z 422.688,A -85,B 0,C 180,E1 -27126.765,E2 -27126.765} C_VEL
LIN {X 0,Y 96.946,Z 409.291,A -85,B 0,C 180,E1 -27130.139,E2 -27130.139} C_VEL
LIN {X 0,Y 97.178,Z 396.636,A -85,B 0,C 180,E1 -27132.537,E2 -27132.537} C_VEL
LIN {X 0,Y 95.917,Z 391.757,A -85,B 0,C 180,E1 -27133.78,E2 -27133.78} C_VEL
LIN {X 0,Y 95.049,Z 388.472,A -85,B 0,C 180,E1 -27138.282,E2 -27138.282} C_VEL
LIN {X 0,Y 93.995,Z 383.847,A -85,B 0,C 180,E1 -27145.484,E2 -27145.484} C_VEL
LIN {X 0,Y 93.672,Z 383.817,A -85,B 0,C 180,E1 -27154.199,E2 -27154.199} C_VEL
LIN {X 0,Y 93.682,Z 383.807,A -85,B 0,C 180,E1 -27157.969,E2 -27157.969} C_VEL
LIN {X 0,Y 94.014,Z 383.759,A -85,B 0,C 180,E1 -27167.04,E2 -27167.04} C_VEL
LIN {X 0,Y 94.159,Z 383.756,A -85,B 0,C 180,E1 -27171.415,E2 -27171.415} C_VEL
LIN {X 0,Y 94.769,Z 383.679,A -85,B 0,C 180,E1 -27180,E2 -27180} C_VEL
LIN {X 0,Y 94.195,Z 383.752,A -85,B 0,C 180,E1 -27188.582,E2 -27188.582} C_VEL
LIN {X 0,Y 94.04,Z 383.763,A -85,B 0,C 180,E1 -27193.707,E2 -27193.707} C_VEL
LIN {X 0,Y 93.69,Z 383.807,A -85,B 0,C 180,E1 -27202.028,E2 -27202.028} C_VEL
LIN {X 0,Y 93.621,Z 383.822,A -85,B 0,C 180,E1 -27206.77,E2 -27206.77} C_VEL
LIN {X 0,Y 93.599,Z 383.827,A -85,B 0,C 180,E1 -27214.317,E2 -27214.317} C_VEL
LIN {X 0,Y 93.546,Z 383.833,A -85,B 0,C 180,E1 -27222.544,E2 -27222.544} C_VEL
LIN {X 0,Y 93.546,Z 383.831,A -85,B 0,C 180,E1 -27228.702,E2 -27228.702} C_VEL
LIN {X 0,Y 93.58,Z 383.821,A -85,B 0,C 180,E1 -27236.219,E2 -27236.219} C_VEL
LIN {X 0,Y 92.917,Z 383.912,A -85,B 0,C 180,E1 -27239.817,E2 -27239.817} C_VEL
LIN {X 0,Y 91.472,Z 384.104,A -85,B 0,C 180,E1 -27243.394,E2 -27243.394} C_VEL
LIN {X 0,Y 87.308,Z 384.627,A -85,B 0,C 180,E1 -27253.396,E2 -27253.396} C_VEL
LIN {X 0,Y 86.968,Z 384.651,A -85,B 0,C 180,E1 -27256.048,E2 -27256.048} C_VEL
LIN {X 0,Y 87.119,Z 384.627,A -85,B 0,C 180,E1 -27260.715,E2 -27260.715} C_VEL
LIN {X 0,Y 87.724,Z 384.559,A -85,B 0,C 180,E1 -27270,E2 -27270} C_VEL
LIN {X 0,Y 87.108,Z 384.635,A -85,B 0,C 180,E1 -27279.286,E2 -27279.286} C_VEL
LIN {X 0,Y 86.951,Z 384.652,A -85,B 0,C 180,E1 -27284.087,E2 -27284.087} C_VEL
LIN {X 0,Y 86.758,Z 384.896,A -85,B 0,C 180,E1 -27289.829,E2 -27289.829} C_VEL
LIN {X 0,Y 87.066,Z 386.137,A -85,B 0,C 180,E1 -27290.68,E2 -27290.68} C_VEL
LIN {X 0,Y 90.416,Z 396.609,A -85,B 0,C 180,E1 -27294.695,E2 -27294.695} C_VEL
LIN {X 0,Y 93.129,Z 406.664,A -85,B 0,C 180,E1 -27298.756,E2 -27298.756} C_VEL
LIN {X 0,Y 94.822,Z 413.786,A -85,B 0,C 180,E1 -27301.89,E2 -27301.89} C_VEL
LIN {X 0,Y 94.468,Z 416.416,A -85,B 0,C 180,E1 -27302.958,E2 -27302.958} C_VEL
LIN {X 0,Y 91.404,Z 428.516,A -85,B 0,C 180,E1 -27308.595,E2 -27308.595} C_VEL
LIN {X 0,Y 89.044,Z 438.736,A -85,B 0,C 180,E1 -27314.737,E2 -27314.737} C_VEL
LIN {X 0,Y 87.356,Z 448.414,A -85,B 0,C 180,E1 -27322.125,E2 -27322.125} C_VEL
LIN {X 0,Y 86.837,Z 456.254,A -85,B 0,C 180,E1 -27329.613,E2 -27329.613} C_VEL
LIN {X 0,Y 87.741,Z 463.029,A -85,B 0,C 180,E1 -27337.637,E2 -27337.637} C_VEL
LIN {X 0,Y 90.705,Z 469.244,A -85,B 0,C 180,E1 -27346.559,E2 -27346.559} C_VEL
LIN {X 0,Y 94.805,Z 473.234,A -85,B 0,C 180,E1 -27353.616,E2 -27353.616} C_VEL
LIN {X 0,Y 100.167,Z 476.11,A -85,B 0,C 180,E1 -27360,E2 -27360} C_VEL
LIN {X 0,Y 105.826,Z 477.802,A -85,B 0,C 180,E1 -27365.04,E2 -27365.04} C_VEL
LIN {X 0,Y 114.535,Z 478.83,A -85,B 0,C 180,E1 -27370.962,E2 -27370.962} C_VEL
LIN {X 0,Y 125.09,Z 478.4,A -85,B 0,C 180,E1 -27376.315,E2 -27376.315} C_VEL
LIN {X 0,Y 134.734,Z 476.781,A -85,B 0,C 180,E1 -27380.134,E2 -27380.134} C_VEL
LIN {X 0,Y 137.117,Z 476.217,A -85,B 0,C 180,E1 -27381.026,E2 -27381.026} C_VEL
LIN {X 0,Y 137.683,Z 476.631,A -85,B 0,C 180,E1 -27383.251,E2 -27383.251} C_VEL
LIN {X 0,Y 137.001,Z 478.208,A -85,B 0,C 180,E1 -27387.496,E2 -27387.496} C_VEL
LIN {X 0,Y 136.516,Z 478.899,A -85,B 0,C 180,E1 -27388.937,E2 -27388.937} C_VEL
LIN {X 0,Y 134.201,Z 480.108,A -85,B 0,C 180,E1 -27390.223,E2 -27390.223} C_VEL
LIN {X 0,Y 126.719,Z 483.501,A -85,B 0,C 180,E1 -27393.706,E2 -27393.706} C_VEL
LIN {X 0,Y 116.736,Z 487.082,A -85,B 0,C 180,E1 -27398.498,E2 -27398.498} C_VEL
LIN {X 0,Y 107.467,Z 489.53,A -85,B 0,C 180,E1 -27403.999,E2 -27403.999} C_VEL
LIN {X 0,Y 99.312,Z 490.818,A -85,B 0,C 180,E1 -27410.44,E2 -27410.44} C_VEL
LIN {X 0,Y 92.867,Z 490.973,A -85,B 0,C 180,E1 -27418.013,E2 -27418.013} C_VEL
LIN {X 0,Y 88.878,Z 490.088,A -85,B 0,C 180,E1 -27426.711,E2 -27426.711} C_VEL
LIN {X 0,Y 87.442,Z 488.023,A -85,B 0,C 180,E1 -27436.048,E2 -27436.048} C_VEL
LIN {X 0,Y 88.545,Z 484.697,A -85,B 0,C 180,E1 -27445.448,E2 -27445.448} C_VEL
LIN {X 0,Y 89.12,Z 483.589,A -85,B 0,C 180,E1 -27447.74,E2 -27447.74} C_VEL
LIN {X 0,Y 88.913,Z 482.093,A -85,B 0,C 180,E1 -27450,E2 -27450} C_VEL
LIN {X 0,Y 87.958,Z 476.281,A -85,B 0,C 180,E1 -27456.883,E2 -27456.883} C_VEL
LIN {X 0,Y 87.992,Z 468.897,A -85,B 0,C 180,E1 -27463.863,E2 -27463.863} C_VEL
LIN {X 0,Y 88.68,Z 462.999,A -85,B 0,C 180,E1 -27468.481,E2 -27468.481} C_VEL
LIN {X 0,Y 88.509,Z 454.211,A -85,B 0,C 180,E1 -27474.013,E2 -27474.013} C_VEL
LIN {X 0,Y 88.636,Z 444.109,A -85,B 0,C 180,E1 -27479.284,E2 -27479.284} C_VEL
LIN {X 0,Y 89.081,Z 432.563,A -85,B 0,C 180,E1 -27484.202,E2 -27484.202} C_VEL
LIN {X 0,Y 89.695,Z 418.779,A -85,B 0,C 180,E1 -27488.816,E2 -27488.816} C_VEL
LIN {X 0,Y 90.239,Z 406.45,A -85,B 0,C 180,E1 -27491.978,E2 -27491.978} C_VEL
LIN {X 0,Y 90.389,Z 397.744,A -85,B 0,C 180,E1 -27493.773,E2 -27493.773} C_VEL
LIN {X 0,Y 88.423,Z 390.788,A -85,B 0,C 180,E1 -27495.669,E2 -27495.669} C_VEL
LIN {X 0,Y 88.014,Z 389.061,A -85,B 0,C 180,E1 -27497.899,E2 -27497.899} C_VEL
LIN {X 0,Y 86.965,Z 384.713,A -85,B 0,C 180,E1 -27505.312,E2 -27505.312} C_VEL
LIN {X 0,Y 86.593,Z 384.698,A -85,B 0,C 180,E1 -27513.221,E2 -27513.221} C_VEL
LIN {X 0,Y 86.617,Z 384.696,A -85,B 0,C 180,E1 -27521.061,E2 -27521.061} C_VEL
LIN {X 0,Y 86.879,Z 384.648,A -85,B 0,C 180,E1 -27526.098,E2 -27526.098} C_VEL
LIN {X 0,Y 87.061,Z 384.637,A -85,B 0,C 180,E1 -27530.709,E2 -27530.709} C_VEL
LIN {X 0,Y 87.699,Z 384.56,A -85,B 0,C 180,E1 -27540,E2 -27540} C_VEL
LIN {X 0,Y 87.104,Z 384.635,A -85,B 0,C 180,E1 -27549.286,E2 -27549.286} C_VEL
LIN {X 0,Y 86.949,Z 384.647,A -85,B 0,C 180,E1 -27554.087,E2 -27554.087} C_VEL
LIN {X 0,Y 86.585,Z 384.697,A -85,B 0,C 180,E1 -27563.944,E2 -27563.944} C_VEL
LIN {X 0,Y 86.477,Z 384.707,A -85,B 0,C 180,E1 -27569.184,E2 -27569.184} C_VEL
LIN {X 0,Y 86.519,Z 384.707,A -85,B 0,C 180,E1 -27575.68,E2 -27575.68} C_VEL
LIN {X 0,Y 86.486,Z 384.711,A -85,B 0,C 180,E1 -27583.002,E2 -27583.002} C_VEL
LIN {X 0,Y 86.466,Z 384.713,A -85,B 0,C 180,E1 -27589.441,E2 -27589.441} C_VEL
LIN {X 0,Y 86.492,Z 384.699,A -85,B 0,C 180,E1 -27596.029,E2 -27596.029} C_VEL
LIN {X 0,Y 86.585,Z 384.691,A -85,B 0,C 180,E1 -27603.234,E2 -27603.234} C_VEL
LIN {X 0,Y 86.649,Z 384.684,A -85,B 0,C 180,E1 -27611.069,E2 -27611.069} C_VEL
LIN {X 0,Y 86.968,Z 384.651,A -85,B 0,C 180,E1 -27616.048,E2 -27616.048} C_VEL
LIN {X 0,Y 86.253,Z 384.735,A -85,B 0,C 180,E1 -27619.934,E2 -27619.934} C_VEL
LIN {X 0,Y 84.726,Z 384.933,A -85,B 0,C 180,E1 -27623.797,E2 -27623.797} C_VEL
LIN {X 0,Y 80.344,Z 385.463,A -85,B 0,C 180,E1 -27634.671,E2 -27634.671} C_VEL
LIN {X 0,Y 79.986,Z 385.503,A -85,B 0,C 180,E1 -27637.575,E2 -27637.575} C_VEL
LIN {X 0,Y 79.85,Z 385.538,A -85,B 0,C 180,E1 -27644.496,E2 -27644.496} C_VEL
LIN {X 0,Y 79.74,Z 385.783,A -85,B 0,C 180,E1 -27647.967,E2 -27647.967} C_VEL
LIN {X 0,Y 80.03,Z 386.956,A -85,B 0,C 180,E1 -27648.894,E2 -27648.894} C_VEL
LIN {X 0,Y 83.216,Z 396.736,A -85,B 0,C 180,E1 -27652.992,E2 -27652.992} C_VEL
LIN {X 0,Y 86.215,Z 407.986,A -85,B 0,C 180,E1 -27657.951,E2 -27657.951} C_VEL
LIN {X 0,Y 87.851,Z 415.035,A -85,B 0,C 180,E1 -27661.331,E2 -27661.331} C_VEL
LIN {X 0,Y 85.082,Z 425.856,A -85,B 0,C 180,E1 -27666.387,E2 -27666.387} C_VEL
LIN {X 0,Y 82.366,Z 436.864,A -85,B 0,C 180,E1 -27673.046,E2 -27673.046} C_VEL
LIN {X 0,Y 80.477,Z 446.728,A -85,B 0,C 180,E1 -27680.721,E2 -27680.721} C_VEL
LIN {X 0,Y 79.78,Z 454.29,A -85,B 0,C 180,E1 -27688.092,E2 -27688.092} C_VEL
LIN {X 0,Y 80.437,Z 461.678,A -85,B 0,C 180,E1 -27696.848,E2 -27696.848} C_VEL
LIN {X 0,Y 82.776,Z 467.625,A -85,B 0,C 180,E1 -27705.244,E2 -27705.244} C_VEL
LIN {X 0,Y 86.826,Z 472.364,A -85,B 0,C 180,E1 -27713.182,E2 -27713.182} C_VEL
LIN {X 0,Y 92.027,Z 475.79,A -85,B 0,C 180,E1 -27720,E2 -27720} C_VEL
LIN {X 0,Y 99.025,Z 478.38,A -85,B 0,C 180,E1 -27726.493,E2 -27726.493} C_VEL
LIN {X 0,Y 108.013,Z 479.886,A -85,B 0,C 180,E1 -27732.587,E2 -27732.587} C_VEL
LIN {X 0,Y 117.998,Z 480.063,A -85,B 0,C 180,E1 -27737.648,E2 -27737.648} C_VEL
LIN {X 0,Y 128.713,Z 478.937,A -85,B 0,C 180,E1 -27741.842,E2 -27741.842} C_VEL
LIN {X 0,Y 129.906,Z 478.716,A -85,B 0,C 180,E1 -27742.254,E2 -27742.254} C_VEL
LIN {X 0,Y 130.744,Z 478.969,A -85,B 0,C 180,E1 -27743.965,E2 -27743.965} C_VEL
LIN {X 0,Y 129.906,Z 480.383,A -85,B 0,C 180,E1 -27747.653,E2 -27747.653} C_VEL
LIN {X 0,Y 122.142,Z 483.461,A -85,B 0,C 180,E1 -27751.189,E2 -27751.189} C_VEL
LIN {X 0,Y 112.42,Z 486.439,A -85,B 0,C 180,E1 -27755.641,E2 -27755.641} C_VEL
LIN {X 0,Y 102.656,Z 488.572,A -85,B 0,C 180,E1 -27761.144,E2 -27761.144} C_VEL
LIN {X 0,Y 93.982,Z 489.574,A -85,B 0,C 180,E1 -27767.7,E2 -27767.7} C_VEL
LIN {X 0,Y 86.979,Z 489.473,A -85,B 0,C 180,E1 -27775.556,E2 -27775.556} C_VEL
LIN {X 0,Y 82.513,Z 488.323,A -85,B 0,C 180,E1 -27784.795,E2 -27784.795} C_VEL
LIN {X 0,Y 80.766,Z 486.043,A -85,B 0,C 180,E1 -27794.868,E2 -27794.868} C_VEL
LIN {X 0,Y 81.778,Z 482.405,A -85,B 0,C 180,E1 -27805.07,E2 -27805.07} C_VEL
LIN {X 0,Y 82.335,Z 481.269,A -85,B 0,C 180,E1 -27807.554,E2 -27807.554} C_VEL
LIN {X 0,Y 81.531,Z 477.725,A -85,B 0,C 180,E1 -27812.47,E2 -27812.47} C_VEL
LIN {X 0,Y 80.934,Z 471.109,A -85,B 0,C 180,E1 -27820.001,E2 -27820.001} C_VEL
LIN {X 0,Y 81.663,Z 462.438,A -85,B 0,C 180,E1 -27827.819,E2 -27827.819} C_VEL
LIN {X 0,Y 81.433,Z 453.147,A -85,B 0,C 180,E1 -27834.201,E2 -27834.201} C_VEL
LIN {X 0,Y 81.601,Z 442.638,A -85,B 0,C 180,E1 -27840.145,E2 -27840.145} C_VEL
LIN {X 0,Y 82.106,Z 431.446,A -85,B 0,C 180,E1 -27845.293,E2 -27845.293} C_VEL
LIN {X 0,Y 82.876,Z 417.759,A -85,B 0,C 180,E1 -27850.251,E2 -27850.251} C_VEL
LIN {X 0,Y 83.6,Z 404.209,A -85,B 0,C 180,E1 -27853.946,E2 -27853.946} C_VEL
LIN {X 0,Y 83.616,Z 399.285,A -85,B 0,C 180,E1 -27855.078,E2 -27855.078} C_VEL
LIN {X 0,Y 80.896,Z 389.538,A -85,B 0,C 180,E1 -27857.995,E2 -27857.995} C_VEL
LIN {X 0,Y 79.941,Z 385.587,A -85,B 0,C 180,E1 -27864.764,E2 -27864.764} C_VEL
LIN {X 0,Y 79.531,Z 385.579,A -85,B 0,C 180,E1 -27873.778,E2 -27873.778} C_VEL
LIN {X 0,Y 79.496,Z 385.577,A -85,B 0,C 180,E1 -27879.29,E2 -27879.29} C_VEL
LIN {X 0,Y 79.781,Z 385.533,A -85,B 0,C 180,E1 -27885.692,E2 -27885.692} C_VEL
LIN {X 0,Y 79.94,Z 385.521,A -85,B 0,C 180,E1 -27889.873,E2 -27889.873} C_VEL
LIN {X 0,Y 80.628,Z 385.441,A -85,B 0,C 180,E1 -27900,E2 -27900} C_VEL
LIN {X 0,Y 79.99,Z 385.521,A -85,B 0,C 180,E1 -27910.121,E2 -27910.121} C_VEL
LIN {X 0,Y 79.761,Z 385.546,A -85,B 0,C 180,E1 -27915.328,E2 -27915.328} C_VEL
LIN {X 0,Y 79.512,Z 385.574,A -85,B 0,C 180,E1 -27920.705,E2 -27920.705} C_VEL
LIN {X 0,Y 79.482,Z 385.582,A -85,B 0,C 180,E1 -27927.846,E2 -27927.846} C_VEL
LIN {X 0,Y 79.385,Z 385.593,A -85,B 0,C 180,E1 -27932.086,E2 -27932.086} C_VEL
LIN {X 0,Y 79.375,Z 385.59,A -85,B 0,C 180,E1 -27938.301,E2 -27938.301} C_VEL
LIN {X 0,Y 79.411,Z 385.588,A -85,B 0,C 180,E1 -27945.074,E2 -27945.074} C_VEL
LIN {X 0,Y 79.393,Z 385.592,A -85,B 0,C 180,E1 -27952.815,E2 -27952.815} C_VEL
LIN {X 0,Y 79.385,Z 385.596,A -85,B 0,C 180,E1 -27957.915,E2 -27957.915} C_VEL
LIN {X 0,Y 79.526,Z 385.571,A -85,B 0,C 180,E1 -27963.778,E2 -27963.778} C_VEL
LIN {X 0,Y 79.515,Z 385.577,A -85,B 0,C 180,E1 -27969.296,E2 -27969.296} C_VEL
LIN {X 0,Y 79.837,Z 385.537,A -85,B 0,C 180,E1 -27976.038,E2 -27976.038} C_VEL
LIN {X 0,Y 80.002,Z 385.511,A -85,B 0,C 180,E1 -27979.881,E2 -27979.881} C_VEL
LIN {X 0,Y 80.652,Z 385.44,A -85,B 0,C 180,E1 -27990,E2 -27990} C_VEL
LIN {X 0,Y 79.986,Z 385.503,A -85,B 0,C 180,E1 -27997.575,E2 -27997.575} C_VEL
LIN {X 0,Y 79.747,Z 386.081,A -85,B 0,C 180,E1 -28000.266,E2 -28000.266} C_VEL
LIN {X 0,Y 79.171,Z 388.01,A -85,B 0,C 180,E1 -28003.412,E2 -28003.412} C_VEL
LIN {X 0,Y 78.499,Z 390.844,A -85,B 0,C 180,E1 -28006.269,E2 -28006.269} C_VEL
LIN {X 0,Y 77.796,Z 395.146,A -85,B 0,C 180,E1 -28009.405,E2 -28009.405} C_VEL
LIN {X 0,Y 77.649,Z 401.654,A -85,B 0,C 180,E1 -28013.184,E2 -28013.184} C_VEL
LIN {X 0,Y 78.222,Z 405.012,A -85,B 0,C 180,E1 -28014.908,E2 -28014.908} C_VEL
LIN {X 0,Y 80.558,Z 414.818,A -85,B 0,C 180,E1 -28019.883,E2 -28019.883} C_VEL
LIN {X 0,Y 80.698,Z 416.331,A -85,B 0,C 180,E1 -28020.66,E2 -28020.66} C_VEL
LIN {X 0,Y 77.65,Z 427.42,A -85,B 0,C 180,E1 -28026.361,E2 -28026.361} C_VEL
LIN {X 0,Y 75.009,Z 437.927,A -85,B 0,C 180,E1 -28033.437,E2 -28033.437} C_VEL
LIN {X 0,Y 73.303,Z 446.889,A -85,B 0,C 180,E1 -28041.061,E2 -28041.061} C_VEL
LIN {X 0,Y 72.718,Z 455.724,A -85,B 0,C 180,E1 -28050.436,E2 -28050.436} C_VEL
LIN {X 0,Y 73.848,Z 462.777,A -85,B 0,C 180,E1 -28059.598,E2 -28059.598} C_VEL
LIN {X 0,Y 77.209,Z 469.266,A -85,B 0,C 180,E1 -28069.511,E2 -28069.511} C_VEL
LIN {X 0,Y 82.022,Z 473.828,A -85,B 0,C 180,E1 -28077.545,E2 -28077.545} C_VEL
LIN {X 0,Y 88.196,Z 477.253,A -85,B 0,C 180,E1 -28084.571,E2 -28084.571} C_VEL
LIN {X 0,Y 92.959,Z 478.938,A -85,B 0,C 180,E1 -28088.697,E2 -28088.697} C_VEL
LIN {X 0,Y 101.609,Z 480.763,A -85,B 0,C 180,E1 -28094.461,E2 -28094.461} C_VEL
LIN {X 0,Y 111.877,Z 481.457,A -85,B 0,C 180,E1 -28099.565,E2 -28099.565} C_VEL
LIN {X 0,Y 122.854,Z 480.857,A -85,B 0,C 180,E1 -28103.756,E2 -28103.756} C_VEL
LIN {X 0,Y 123.675,Z 480.917,A -85,B 0,C 180,E1 -28104.605,E2 -28104.605} C_VEL
LIN {X 0,Y 121.95,Z 481.961,A -85,B 0,C 180,E1 -28106.716,E2 -28106.716} C_VEL
LIN {X 0,Y 113.813,Z 484.42,A -85,B 0,C 180,E1 -28110.176,E2 -28110.176} C_VEL
LIN {X 0,Y 103.132,Z 486.765,A -85,B 0,C 180,E1 -28115.142,E2 -28115.142} C_VEL
LIN {X 0,Y 93.362,Z 488.031,A -85,B 0,C 180,E1 -28121.171,E2 -28121.171} C_VEL
LIN {X 0,Y 84.841,Z 488.169,A -85,B 0,C 180,E1 -28128.495,E2 -28128.495} C_VEL
LIN {X 0,Y 78.47,Z 487.278,A -85,B 0,C 180,E1 -28137.496,E2 -28137.496} C_VEL
LIN {X 0,Y 74.839,Z 485.305,A -85,B 0,C 180,E1 -28147.937,E2 -28147.937} C_VEL
LIN {X 0,Y 74.235,Z 482.176,A -85,B 0,C 180,E1 -28159.086,E2 -28159.086} C_VEL
LIN {X 0,Y 75.049,Z 480.079,A -85,B 0,C 180,E1 -28164.627,E2 -28164.627} C_VEL
LIN {X 0,Y 75.511,Z 478.782,A -85,B 0,C 180,E1 -28167.333,E2 -28167.333} C_VEL
LIN {X 0,Y 74.502,Z 473.979,A -85,B 0,C 180,E1 -28174.057,E2 -28174.057} C_VEL
LIN {X 0,Y 74.144,Z 466.659,A -85,B 0,C 180,E1 -28182.314,E2 -28182.314} C_VEL
LIN {X 0,Y 74.668,Z 460.645,A -85,B 0,C 180,E1 -28187.927,E2 -28187.927} C_VEL
LIN {X 0,Y 74.337,Z 450.817,A -85,B 0,C 180,E1 -28195.178,E2 -28195.178} C_VEL
LIN {X 0,Y 74.631,Z 440.097,A -85,B 0,C 180,E1 -28201.64,E2 -28201.64} C_VEL
LIN {X 0,Y 75.237,Z 428.21,A -85,B 0,C 180,E1 -28207.384,E2 -28207.384} C_VEL
LIN {X 0,Y 76.103,Z 416.332,A -85,B 0,C 180,E1 -28211.941,E2 -28211.941} C_VEL
LIN {X 0,Y 76.938,Z 402.956,A -85,B 0,C 180,E1 -28215.854,E2 -28215.854} C_VEL
LIN {X 0,Y 76.74,Z 400.283,A -85,B 0,C 180,E1 -28216.621,E2 -28216.621} C_VEL
LIN {X 0,Y 73.944,Z 390.817,A -85,B 0,C 180,E1 -28219.69,E2 -28219.69} C_VEL
LIN {X 0,Y 73.331,Z 388.242,A -85,B 0,C 180,E1 -28220.826,E2 -28220.826} C_VEL
LIN {X 0,Y 72.926,Z 386.433,A -85,B 0,C 180,E1 -28224.264,E2 -28224.264} C_VEL
LIN {X 0,Y 72.476,Z 386.451,A -85,B 0,C 180,E1 -28230.997,E2 -28230.997} C_VEL
LIN {X 0,Y 72.387,Z 386.458,A -85,B 0,C 180,E1 -28237.147,E2 -28237.147} C_VEL
LIN {X 0,Y 72.678,Z 386.419,A -85,B 0,C 180,E1 -28245.236,E2 -28245.236} C_VEL
LIN {X 0,Y 72.828,Z 386.402,A -85,B 0,C 180,E1 -28248.872,E2 -28248.872} C_VEL
LIN {X 0,Y 73.555,Z 386.322,A -85,B 0,C 180,E1 -28260,E2 -28260} C_VEL
LIN {X 0,Y 72.877,Z 386.405,A -85,B 0,C 180,E1 -28271.12,E2 -28271.12} C_VEL
LIN {X 0,Y 72.581,Z 386.444,A -85,B 0,C 180,E1 -28276.887,E2 -28276.887} C_VEL
LIN {X 0,Y 72.393,Z 386.461,A -85,B 0,C 180,E1 -28282.85,E2 -28282.85} C_VEL
LIN {X 0,Y 72.376,Z 386.462,A -85,B 0,C 180,E1 -28289.083,E2 -28289.083} C_VEL
LIN {X 0,Y 72.301,Z 386.477,A -85,B 0,C 180,E1 -28295.678,E2 -28295.678} C_VEL
LIN {X 0,Y 72.262,Z 386.483,A -85,B 0,C 180,E1 -28302.906,E2 -28302.906} C_VEL
LIN {X 0,Y 72.301,Z 386.479,A -85,B 0,C 180,E1 -28311.045,E2 -28311.045} C_VEL
LIN {X 0,Y 72.3,Z 386.471,A -85,B 0,C 180,E1 -28314.323,E2 -28314.323} C_VEL
LIN {X 0,Y 72.392,Z 386.464,A -85,B 0,C 180,E1 -28320.961,E2 -28320.961} C_VEL
LIN {X 0,Y 72.395,Z 386.467,A -85,B 0,C 180,E1 -28327.151,E2 -28327.151} C_VEL
LIN {X 0,Y 72.737,Z 386.424,A -85,B 0,C 180,E1 -28335.066,E2 -28335.066} C_VEL
LIN {X 0,Y 72.886,Z 386.398,A -85,B 0,C 180,E1 -28338.881,E2 -28338.881} C_VEL
LIN {X 0,Y 73.578,Z 386.321,A -85,B 0,C 180,E1 -28350,E2 -28350} C_VEL
LIN {X 0,Y 72.883,Z 386.399,A -85,B 0,C 180,E1 -28361.119,E2 -28361.119} C_VEL
LIN {X 0,Y 72.772,Z 386.669,A -85,B 0,C 180,E1 -28365.857,E2 -28365.857} C_VEL
LIN {X 0,Y 72.989,Z 387.796,A -85,B 0,C 180,E1 -28366.79,E2 -28366.79} C_VEL
LIN {X 0,Y 76.321,Z 398.068,A -85,B 0,C 180,E1 -28371.613,E2 -28371.613} C_VEL
LIN {X 0,Y 78.222,Z 405.012,A -85,B 0,C 180,E1 -28374.908,E2 -28374.908} C_VEL
LIN {X 0,Y 78.285,Z 408.399,A -85,B 0,C 180,E1 -28376.396,E2 -28376.396} C_VEL
LIN {X 0,Y 77.247,Z 411.773,A -85,B 0,C 180,E1 -28377.734,E2 -28377.734} C_VEL
LIN {X 0,Y 72.257,Z 421.57,A -85,B 0,C 180,E1 -28382.032,E2 -28382.032} C_VEL
LIN {X 0,Y 71.917,Z 422.669,A -85,B 0,C 180,E1 -28382.635,E2 -28382.635} C_VEL
LIN {X 0,Y 69.057,Z 433.023,A -85,B 0,C 180,E1 -28389.247,E2 -28389.247} C_VEL
LIN {X 0,Y 66.838,Z 442.879,A -85,B 0,C 180,E1 -28397.394,E2 -28397.394} C_VEL
LIN {X 0,Y 65.746,Z 451.059,A -85,B 0,C 180,E1 -28405.861,E2 -28405.861} C_VEL
LIN {X 0,Y 66.116,Z 459.395,A -85,B 0,C 180,E1 -28416.428,E2 -28416.428} C_VEL
LIN {X 0,Y 68.598,Z 466.225,A -85,B 0,C 180,E1 -28426.673,E2 -28426.673} C_VEL
LIN {X 0,Y 73.86,Z 472.468,A -85,B 0,C 180,E1 -28437.273,E2 -28437.273} C_VEL
LIN {X 0,Y 80.06,Z 476.54,A -85,B 0,C 180,E1 -28445.036,E2 -28445.036} C_VEL
LIN {X 0,Y 85.66,Z 478.916,A -85,B 0,C 180,E1 -28450.095,E2 -28450.095} C_VEL
LIN {X 0,Y 96.067,Z 481.588,A -85,B 0,C 180,E1 -28457.016,E2 -28457.016} C_VEL
LIN {X 0,Y 105.951,Z 482.662,A -85,B 0,C 180,E1 -28461.778,E2 -28461.778} C_VEL
LIN {X 0,Y 108.626,Z 482.724,A -85,B 0,C 180,E1 -28462.842,E2 -28462.842} C_VEL
LIN {X 0,Y 113.561,Z 483.008,A -85,B 0,C 180,E1 -28465.672,E2 -28465.672} C_VEL
LIN {X 0,Y 104.727,Z 484.95,A -85,B 0,C 180,E1 -28469.264,E2 -28469.264} C_VEL
LIN {X 0,Y 93.92,Z 486.44,A -85,B 0,C 180,E1 -28474.604,E2 -28474.604} C_VEL
LIN {X 0,Y 84.101,Z 486.839,A -85,B 0,C 180,E1 -28481.229,E2 -28481.229} C_VEL
LIN {X 0,Y 75.87,Z 486.166,A -85,B 0,C 180,E1 -28489.578,E2 -28489.578} C_VEL
LIN {X 0,Y 70.202,Z 484.478,A -85,B 0,C 180,E1 -28499.964,E2 -28499.964} C_VEL
LIN {X 0,Y 67.622,Z 481.673,A -85,B 0,C 180,E1 -28511.833,E2 -28511.833} C_VEL
LIN {X 0,Y 68.387,Z 477.615,A -85,B 0,C 180,E1 -28524.102,E2 -28524.102} C_VEL
LIN {X 0,Y 68.66,Z 476.249,A -85,B 0,C 180,E1 -28527.066,E2 -28527.066} C_VEL
LIN {X 0,Y 67.548,Z 471.102,A -85,B 0,C 180,E1 -28534.475,E2 -28534.475} C_VEL
LIN {X 0,Y 67.361,Z 463.352,A -85,B 0,C 180,E1 -28543.577,E2 -28543.577} C_VEL
LIN {X 0,Y 67.669,Z 460.394,A -85,B 0,C 180,E1 -28546.595,E2 -28546.595} C_VEL
LIN {X 0,Y 67.311,Z 452.313,A -85,B 0,C 180,E1 -28553.422,E2 -28553.422} C_VEL
LIN {X 0,Y 67.423,Z 442.156,A -85,B 0,C 180,E1 -28560.54,E2 -28560.54} C_VEL
LIN {X 0,Y 68.085,Z 430.905,A -85,B 0,C 180,E1 -28566.973,E2 -28566.973} C_VEL
LIN {X 0,Y 69.031,Z 418.865,A -85,B 0,C 180,E1 -28572.413,E2 -28572.413} C_VEL
LIN {X 0,Y 70.084,Z 405.585,A -85,B 0,C 180,E1 -28577.029,E2 -28577.029} C_VEL
LIN {X 0,Y 70.232,Z 402.594,A -85,B 0,C 180,E1 -28577.906,E2 -28577.906} C_VEL
LIN {X 0,Y 67.047,Z 391.058,A -85,B 0,C 180,E1 -28582.225,E2 -28582.225} C_VEL
LIN {X 0,Y 66.01,Z 387.87,A -85,B 0,C 180,E1 -28583.684,E2 -28583.684} C_VEL
LIN {X 0,Y 65.788,Z 387.331,A -85,B 0,C 180,E1 -28584.956,E2 -28584.956} C_VEL
LIN {X 0,Y 65.281,Z 387.353,A -85,B 0,C 180,E1 -28594.492,E2 -28594.492} C_VEL
LIN {X 0,Y 65.588,Z 387.304,A -85,B 0,C 180,E1 -28604.656,E2 -28604.656} C_VEL
LIN {X 0,Y 65.721,Z 387.282,A -85,B 0,C 180,E1 -28607.65,E2 -28607.65} C_VEL
LIN {X 0,Y 66.48,Z 387.203,A -85,B 0,C 180,E1 -28620,E2 -28620} C_VEL
LIN {X 0,Y 65.771,Z 387.285,A -85,B 0,C 180,E1 -28632.34,E2 -28632.34} C_VEL
LIN {X 0,Y 65.384,Z 387.339,A -85,B 0,C 180,E1 -28638.812,E2 -28638.812} C_VEL
LIN {X 0,Y 65.238,Z 387.359,A -85,B 0,C 180,E1 -28645.525,E2 -28645.525} C_VEL
LIN {X 0,Y 65.198,Z 387.362,A -85,B 0,C 180,E1 -28652.614,E2 -28652.614} C_VEL
LIN {X 0,Y 65.195,Z 387.363,A -85,B 0,C 180,E1 -28661.011,E2 -28661.011} C_VEL
LIN {X 0,Y 65.212,Z 387.361,A -85,B 0,C 180,E1 -28669.713,E2 -28669.713} C_VEL
LIN {X 0,Y 65.254,Z 387.357,A -85,B 0,C 180,E1 -28679.498,E2 -28679.498} C_VEL
LIN {X 0,Y 65.246,Z 387.352,A -85,B 0,C 180,E1 -28684.479,E2 -28684.479} C_VEL
LIN {X 0,Y 65.637,Z 387.309,A -85,B 0,C 180,E1 -28694.507,E2 -28694.507} C_VEL
LIN {X 0,Y 65.777,Z 387.287,A -85,B 0,C 180,E1 -28697.661,E2 -28697.661} C_VEL
LIN {X 0,Y 66.502,Z 387.202,A -85,B 0,C 180,E1 -28710,E2 -28710} C_VEL
LIN {X 0,Y 65.768,Z 387.328,A -85,B 0,C 180,E1 -28722.644,E2 -28722.644} C_VEL
LIN {X 0,Y 65.936,Z 388.283,A -85,B 0,C 180,E1 -28724.135,E2 -28724.135} C_VEL
LIN {X 0,Y 69.669,Z 400.064,A -85,B 0,C 180,E1 -28730.366,E2 -28730.366} C_VEL
LIN {X 0,Y 72.171,Z 409.81,A -85,B 0,C 180,E1 -28735.602,E2 -28735.602} C_VEL
LIN {X 0,Y 73.638,Z 416.834,A -85,B 0,C 180,E1 -28739.598,E2 -28739.598} C_VEL
LIN {X 0,Y 71.917,Z 422.669,A -85,B 0,C 180,E1 -28742.635,E2 -28742.635} C_VEL
LIN {X 0,Y 70.059,Z 427.243,A -85,B 0,C 180,E1 -28745.242,E2 -28745.242} C_VEL
LIN {X 0,Y 65.349,Z 434.169,A -85,B 0,C 180,E1 -28749.738,E2 -28749.738} C_VEL
LIN {X 0,Y 60.823,Z 440.687,A -85,B 0,C 180,E1 -28755.272,E2 -28755.272} C_VEL
LIN {X 0,Y 59.361,Z 444.603,A -85,B 0,C 180,E1 -28759.307,E2 -28759.307} C_VEL
LIN {X 0,Y 58.628,Z 452.898,A -85,B 0,C 180,E1 -28769.187,E2 -28769.187} C_VEL
LIN {X 0,Y 59.655,Z 460.819,A -85,B 0,C 180,E1 -28780.47,E2 -28780.47} C_VEL
LIN {X 0,Y 62.459,Z 466.823,A -85,B 0,C 180,E1 -28790.225,E2 -28790.225} C_VEL
LIN {X 0,Y 69.142,Z 473.552,A -85,B 0,C 180,E1 -28802.131,E2 -28802.131} C_VEL
LIN {X 0,Y 76.928,Z 478.01,A -85,B 0,C 180,E1 -28810.528,E2 -28810.528} C_VEL
LIN {X 0,Y 82.394,Z 480.074,A -85,B 0,C 180,E1 -28814.827,E2 -28814.827} C_VEL
LIN {X 0,Y 89.229,Z 481.933,A -85,B 0,C 180,E1 -28819.067,E2 -28819.067} C_VEL
LIN {X 0,Y 101.167,Z 483.714,A -85,B 0,C 180,E1 -28824.634,E2 -28824.634} C_VEL
LIN {X 0,Y 101.42,Z 484.02,A -85,B 0,C 180,E1 -28825.733,E2 -28825.733} C_VEL
LIN {X 0,Y 90.09,Z 485.19,A -85,B 0,C 180,E1 -28830.896,E2 -28830.896} C_VEL
LIN {X 0,Y 79.662,Z 485.3,A -85,B 0,C 180,E1 -28837.441,E2 -28837.441} C_VEL
LIN {X 0,Y 70.726,Z 484.344,A -85,B 0,C 180,E1 -28845.928,E2 -28845.928} C_VEL
LIN {X 0,Y 64.327,Z 482.393,A -85,B 0,C 180,E1 -28856.889,E2 -28856.889} C_VEL
LIN {X 0,Y 61.193,Z 479.377,A -85,B 0,C 180,E1 -28869.846,E2 -28869.846} C_VEL
LIN {X 0,Y 61.773,Z 475.058,A -85,B 0,C 180,E1 -28883.467,E2 -28883.467} C_VEL
LIN {X 0,Y 61.84,Z 473.473,A -85,B 0,C 180,E1 -28886.743,E2 -28886.743} C_VEL
LIN {X 0,Y 60.52,Z 466.802,A -85,B 0,C 180,E1 -28896.668,E2 -28896.668} C_VEL
LIN {X 0,Y 60.644,Z 459.908,A -85,B 0,C 180,E1 -28905.114,E2 -28905.114} C_VEL
LIN {X 0,Y 60.323,Z 453.625,A -85,B 0,C 180,E1 -28911.244,E2 -28911.244} C_VEL
LIN {X 0,Y 60.309,Z 443.391,A -85,B 0,C 180,E1 -28919.686,E2 -28919.686} C_VEL
LIN {X 0,Y 60.99,Z 431.798,A -85,B 0,C 180,E1 -28927.334,E2 -28927.334} C_VEL
LIN {X 0,Y 62.112,Z 419.392,A -85,B 0,C 180,E1 -28933.785,E2 -28933.785} C_VEL
LIN {X 0,Y 63.408,Z 405.926,A -85,B 0,C 180,E1 -28939.043,E2 -28939.043} C_VEL
LIN {X 0,Y 63.37,Z 403.295,A -85,B 0,C 180,E1 -28940.017,E2 -28940.017} C_VEL
LIN {X 0,Y 60.139,Z 391.7,A -85,B 0,C 180,E1 -28945.128,E2 -28945.128} C_VEL
LIN {X 0,Y 58.683,Z 388.941,A -85,B 0,C 180,E1 -28946.963,E2 -28946.963} C_VEL
LIN {X 0,Y 58.467,Z 388.244,A -85,B 0,C 180,E1 -28948.463,E2 -28948.463} C_VEL
LIN {X 0,Y 58.185,Z 388.228,A -85,B 0,C 180,E1 -28958.754,E2 -28958.754} C_VEL
LIN {X 0,Y 58.597,Z 388.169,A -85,B 0,C 180,E1 -28966.121,E2 -28966.121} C_VEL
LIN {X 0,Y 58.78,Z 388.163,A -85,B 0,C 180,E1 -28973.133,E2 -28973.133} C_VEL
LIN {X 0,Y 59.369,Z 388.089,A -85,B 0,C 180,E1 -28980,E2 -28980} C_VEL
LIN {X 0,Y 58.812,Z 388.154,A -85,B 0,C 180,E1 -28986.863,E2 -28986.863} C_VEL
LIN {X 0,Y 58.524,Z 388.193,A -85,B 0,C 180,E1 -28996.123,E2 -28996.123} C_VEL
LIN {X 0,Y 58.15,Z 388.234,A -85,B 0,C 180,E1 -29008.91,E2 -29008.91} C_VEL
LIN {X 0,Y 58.159,Z 388.237,A -85,B 0,C 180,E1 -29012.235,E2 -29012.235} C_VEL
LIN {X 0,Y 58.038,Z 388.248,A -85,B 0,C 180,E1 -29017.262,E2 -29017.262} C_VEL
LIN {X 0,Y 58.022,Z 388.249,A -85,B 0,C 180,E1 -29026.615,E2 -29026.615} C_VEL
LIN {X 0,Y 58.037,Z 388.251,A -85,B 0,C 180,E1 -29032.738,E2 -29032.738} C_VEL
LIN {X 0,Y 58.153,Z 388.236,A -85,B 0,C 180,E1 -29041.092,E2 -29041.092} C_VEL
LIN {X 0,Y 58.526,Z 388.193,A -85,B 0,C 180,E1 -29053.876,E2 -29053.876} C_VEL
LIN {X 0,Y 58.826,Z 388.158,A -85,B 0,C 180,E1 -29063.139,E2 -29063.139} C_VEL
LIN {X 0,Y 59.394,Z 388.088,A -85,B 0,C 180,E1 -29070,E2 -29070} C_VEL
LIN {X 0,Y 58.74,Z 388.313,A -85,B 0,C 180,E1 -29079.903,E2 -29079.903} C_VEL
LIN {X 0,Y 58.958,Z 389.264,A -85,B 0,C 180,E1 -29081.169,E2 -29081.169} C_VEL
LIN {X 0,Y 62.455,Z 399.909,A -85,B 0,C 180,E1 -29087.647,E2 -29087.647} C_VEL
LIN {X 0,Y 64.754,Z 408.932,A -85,B 0,C 180,E1 -29093.047,E2 -29093.047} C_VEL
LIN {X 0,Y 66.558,Z 417.412,A -85,B 0,C 180,E1 -29098.369,E2 -29098.369} C_VEL
LIN {X 0,Y 63.17,Z 428.927,A -85,B 0,C 180,E1 -29105.421,E2 -29105.421} C_VEL
LIN {X 0,Y 60.581,Z 438.626,A -85,B 0,C 180,E1 -29113.311,E2 -29113.311} C_VEL
LIN {X 0,Y 59.361,Z 444.603,A -85,B 0,C 180,E1 -29119.307,E2 -29119.307} C_VEL
LIN {X 0,Y 58.158,Z 448.382,A -85,B 0,C 180,E1 -29123.58,E2 -29123.58} C_VEL
LIN {X 0,Y 55.088,Z 454.001,A -85,B 0,C 180,E1 -29131.261,E2 -29131.261} C_VEL
LIN {X 0,Y 53.086,Z 459.136,A -85,B 0,C 180,E1 -29140.064,E2 -29140.064} C_VEL
LIN {X 0,Y 53.56,Z 462.163,A -85,B 0,C 180,E1 -29145.532,E2 -29145.532} C_VEL
LIN {X 0,Y 57.91,Z 468.792,A -85,B 0,C 180,E1 -29157.189,E2 -29157.189} C_VEL
LIN {X 0,Y 63.875,Z 473.892,A -85,B 0,C 180,E1 -29166.317,E2 -29166.317} C_VEL
LIN {X 0,Y 72.795,Z 478.672,A -85,B 0,C 180,E1 -29175.111,E2 -29175.111} C_VEL
LIN {X 0,Y 83.342,Z 482.234,A -85,B 0,C 180,E1 -29181.94,E2 -29181.94} C_VEL
LIN {X 0,Y 89.011,Z 483.498,A -85,B 0,C 180,E1 -29184.684,E2 -29184.684} C_VEL
LIN {X 0,Y 86.678,Z 483.868,A -85,B 0,C 180,E1 -29186.89,E2 -29186.89} C_VEL
LIN {X 0,Y 75.622,Z 483.688,A -85,B 0,C 180,E1 -29193.238,E2 -29193.238} C_VEL
LIN {X 0,Y 65.935,Z 482.434,A -85,B 0,C 180,E1 -29201.745,E2 -29201.745} C_VEL
LIN {X 0,Y 58.709,Z 480.236,A -85,B 0,C 180,E1 -29213.235,E2 -29213.235} C_VEL
LIN {X 0,Y 54.918,Z 476.908,A -85,B 0,C 180,E1 -29227.424,E2 -29227.424} C_VEL
LIN {X 0,Y 55.2,Z 472.371,A -85,B 0,C 180,E1 -29242.686,E2 -29242.686} C_VEL
LIN {X 0,Y 55.024,Z 470.611,A -85,B 0,C 180,E1 -29246.339,E2 -29246.339} C_VEL
LIN {X 0,Y 53.649,Z 463.45,A -85,B 0,C 180,E1 -29257.527,E2 -29257.527} C_VEL
LIN {X 0,Y 53.726,Z 457.658,A -85,B 0,C 180,E1 -29265.166,E2 -29265.166} C_VEL
LIN {X 0,Y 53.164,Z 448.817,A -85,B 0,C 180,E1 -29274.399,E2 -29274.399} C_VEL
LIN {X 0,Y 53.514,Z 437.742,A -85,B 0,C 180,E1 -29283.927,E2 -29283.927} C_VEL
LIN {X 0,Y 54.63,Z 424.966,A -85,B 0,C 180,E1 -29292.484,E2 -29292.484} C_VEL
LIN {X 0,Y 56.041,Z 412.652,A -85,B 0,C 180,E1 -29298.801,E2 -29298.801} C_VEL
LIN {X 0,Y 56.824,Z 405.291,A -85,B 0,C 180,E1 -29301.8,E2 -29301.8} C_VEL
LIN {X 0,Y 54.231,Z 395.321,A -85,B 0,C 180,E1 -29307.079,E2 -29307.079} C_VEL
LIN {X 0,Y 51.318,Z 389.767,A -85,B 0,C 180,E1 -29311.358,E2 -29311.358} C_VEL
LIN {X 0,Y 51.125,Z 389.141,A -85,B 0,C 180,E1 -29313.463,E2 -29313.463} C_VEL
LIN {X 0,Y 51.41,Z 389.07,A -85,B 0,C 180,E1 -29324.132,E2 -29324.132} C_VEL
LIN {X 0,Y 51.655,Z 389.051,A -85,B 0,C 180,E1 -29332.18,E2 -29332.18} C_VEL
LIN {X 0,Y 52.252,Z 388.975,A -85,B 0,C 180,E1 -29340,E2 -29340} C_VEL
LIN {X 0,Y 51.688,Z 389.044,A -85,B 0,C 180,E1 -29347.814,E2 -29347.814} C_VEL
LIN {X 0,Y 51.392,Z 389.083,A -85,B 0,C 180,E1 -29356.816,E2 -29356.816} C_VEL
LIN {X 0,Y 51.023,Z 389.127,A -85,B 0,C 180,E1 -29364.407,E2 -29364.407} C_VEL
LIN {X 0,Y 51.032,Z 389.129,A -85,B 0,C 180,E1 -29374.281,E2 -29374.281} C_VEL
LIN {X 0,Y 50.989,Z 389.125,A -85,B 0,C 180,E1 -29386.437,E2 -29386.437} C_VEL
LIN {X 0,Y 51.053,Z 389.12,A -85,B 0,C 180,E1 -29396.59,E2 -29396.59} C_VEL
LIN {X 0,Y 51.027,Z 389.126,A -85,B 0,C 180,E1 -29405.595,E2 -29405.595} C_VEL
LIN {X 0,Y 51.467,Z 389.072,A -85,B 0,C 180,E1 -29414.151,E2 -29414.151} C_VEL
LIN {X 0,Y 51.699,Z 389.042,A -85,B 0,C 180,E1 -29422.187,E2 -29422.187} C_VEL
LIN {X 0,Y 52.279,Z 388.974,A -85,B 0,C 180,E1 -29430,E2 -29430} C_VEL
LIN {X 0,Y 51.829,Z 389.305,A -85,B 0,C 180,E1 -29436.325,E2 -29436.325} C_VEL
LIN {X 0,Y 52.106,Z 390.588,A -85,B 0,C 180,E1 -29437.751,E2 -29437.751} C_VEL
LIN {X 0,Y 54.668,Z 397.801,A -85,B 0,C 180,E1 -29443.001,E2 -29443.001} C_VEL
LIN {X 0,Y 56.993,Z 406.426,A -85,B 0,C 180,E1 -29448.886,E2 -29448.886} C_VEL
LIN {X 0,Y 59.416,Z 417.141,A -85,B 0,C 180,E1 -29456.331,E2 -29456.331} C_VEL
LIN {X 0,Y 59.029,Z 419.503,A -85,B 0,C 180,E1 -29457.835,E2 -29457.835} C_VEL
LIN {X 0,Y 55.436,Z 431.062,A -85,B 0,C 180,E1 -29466.08,E2 -29466.08} C_VEL
LIN {X 0,Y 52.856,Z 441.092,A -85,B 0,C 180,E1 -29475.728,E2 -29475.728} C_VEL
LIN {X 0,Y 51.63,Z 450.265,A -85,B 0,C 180,E1 -29487.011,E2 -29487.011} C_VEL
LIN {X 0,Y 52.384,Z 458.81,A -85,B 0,C 180,E1 -29499.905,E2 -29499.905} C_VEL
LIN {X 0,Y 53.56,Z 462.163,A -85,B 0,C 180,E1 -29505.532,E2 -29505.532} C_VEL
LIN {X 0,Y 54.502,Z 465.078,A -85,B 0,C 180,E1 -29510.909,E2 -29510.909} C_VEL
LIN {X 0,Y 55.499,Z 469.344,A -85,B 0,C 180,E1 -29520.183,E2 -29520.183} C_VEL
LIN {X 0,Y 58.006,Z 473.185,A -85,B 0,C 180,E1 -29529.087,E2 -29529.087} C_VEL
LIN {X 0,Y 61.072,Z 475.373,A -85,B 0,C 180,E1 -29533.479,E2 -29533.479} C_VEL
LIN {X 0,Y 69.834,Z 479.581,A -85,B 0,C 180,E1 -29540.624,E2 -29540.624} C_VEL
LIN {X 0,Y 77.781,Z 482.346,A -85,B 0,C 180,E1 -29545.373,E2 -29545.373} C_VEL
LIN {X 0,Y 66.607,Z 481.34,A -85,B 0,C 180,E1 -29552.425,E2 -29552.425} C_VEL
LIN {X 0,Y 57.144,Z 479.328,A -85,B 0,C 180,E1 -29562.446,E2 -29562.446} C_VEL
LIN {X 0,Y 50.41,Z 476.198,A -85,B 0,C 180,E1 -29576.774,E2 -29576.774} C_VEL
LIN {X 0,Y 48.16,Z 472.142,A -85,B 0,C 180,E1 -29593.031,E2 -29593.031} C_VEL
LIN {X 0,Y 48.685,Z 469.563,A -85,B 0,C 180,E1 -29601.7,E2 -29601.7} C_VEL
LIN {X 0,Y 48.224,Z 467.637,A -85,B 0,C 180,E1 -29605.821,E2 -29605.821} C_VEL
LIN {X 0,Y 46.833,Z 460.012,A -85,B 0,C 180,E1 -29618.63,E2 -29618.63} C_VEL
LIN {X 0,Y 46.846,Z 457.061,A -85,B 0,C 180,E1 -29623.005,E2 -29623.005} C_VEL
LIN {X 0,Y 46.128,Z 448.883,A -85,B 0,C 180,E1 -29632.996,E2 -29632.996} C_VEL
LIN {X 0,Y 46.342,Z 438.723,A -85,B 0,C 180,E1 -29643.349,E2 -29643.349} C_VEL
LIN {X 0,Y 47.446,Z 427.235,A -85,B 0,C 180,E1 -29652.727,E2 -29652.727} C_VEL
LIN {X 0,Y 49.155,Z 414.563,A -85,B 0,C 180,E1 -29660.533,E2 -29660.533} C_VEL
LIN {X 0,Y 50.115,Z 406.251,A -85,B 0,C 180,E1 -29664.657,E2 -29664.657} C_VEL
LIN {X 0,Y 48.269,Z 398.744,A -85,B 0,C 180,E1 -29669.362,E2 -29669.362} C_VEL
LIN {X 0,Y 44.191,Z 390.92,A -85,B 0,C 180,E1 -29676.572,E2 -29676.572} C_VEL
LIN {X 0,Y 44.044,Z 390.035,A -85,B 0,C 180,E1 -29678.959,E2 -29678.959} C_VEL
LIN {X 0,Y 44.19,Z 389.977,A -85,B 0,C 180,E1 -29682.594,E2 -29682.594} C_VEL
LIN {X 0,Y 44.503,Z 389.936,A -85,B 0,C 180,E1 -29690.913,E2 -29690.913} C_VEL
LIN {X 0,Y 45.125,Z 389.862,A -85,B 0,C 180,E1 -29700,E2 -29700} C_VEL
LIN {X 0,Y 44.539,Z 389.937,A -85,B 0,C 180,E1 -29709.079,E2 -29709.079} C_VEL
LIN {X 0,Y 44.155,Z 389.984,A -85,B 0,C 180,E1 -29718.562,E2 -29718.562} C_VEL
LIN {X 0,Y 43.844,Z 390.016,A -85,B 0,C 180,E1 -29728.743,E2 -29728.743} C_VEL
LIN {X 0,Y 43.807,Z 390.021,A -85,B 0,C 180,E1 -29739.92,E2 -29739.92} C_VEL
LIN {X 0,Y 43.845,Z 390.016,A -85,B 0,C 180,E1 -29753.27,E2 -29753.27} C_VEL
LIN {X 0,Y 43.845,Z 390.017,A -85,B 0,C 180,E1 -29761.258,E2 -29761.258} C_VEL
LIN {X 0,Y 44.232,Z 389.967,A -85,B 0,C 180,E1 -29772.426,E2 -29772.426} C_VEL
LIN {X 0,Y 44.548,Z 389.927,A -85,B 0,C 180,E1 -29780.923,E2 -29780.923} C_VEL
LIN {X 0,Y 45.127,Z 390.041,A -85,B 0,C 180,E1 -29790.837,E2 -29790.837} C_VEL
LIN {X 0,Y 45.279,Z 391.362,A -85,B 0,C 180,E1 -29792.78,E2 -29792.78} C_VEL
LIN {X 0,Y 47.984,Z 398.903,A -85,B 0,C 180,E1 -29799.484,E2 -29799.484} C_VEL
LIN {X 0,Y 50.407,Z 408.586,A -85,B 0,C 180,E1 -29807.234,E2 -29807.234} C_VEL
LIN {X 0,Y 52.193,Z 416.788,A -85,B 0,C 180,E1 -29813.825,E2 -29813.825} C_VEL
LIN {X 0,Y 52.46,Z 418.504,A -85,B 0,C 180,E1 -29815.203,E2 -29815.203} C_VEL
LIN {X 0,Y 48.669,Z 430.013,A -85,B 0,C 180,E1 -29824.019,E2 -29824.019} C_VEL
LIN {X 0,Y 45.852,Z 440.346,A -85,B 0,C 180,E1 -29834.854,E2 -29834.854} C_VEL
LIN {X 0,Y 44.585,Z 450.522,A -85,B 0,C 180,E1 -29849.217,E2 -29849.217} C_VEL
LIN {X 0,Y 46.018,Z 459.474,A -85,B 0,C 180,E1 -29864.499,E2 -29864.499} C_VEL
LIN {X 0,Y 50.306,Z 466.75,A -85,B 0,C 180,E1 -29877.885,E2 -29877.885} C_VEL
LIN {X 0,Y 58.87,Z 474.033,A -85,B 0,C 180,E1 -29891.085,E2 -29891.085} C_VEL
LIN {X 0,Y 61.072,Z 475.373,A -85,B 0,C 180,E1 -29893.479,E2 -29893.479} C_VEL
LIN {X 0,Y 62.074,Z 476.226,A -85,B 0,C 180,E1 -29895.454,E2 -29895.454} C_VEL
LIN {X 0,Y 62.077,Z 477.073,A -85,B 0,C 180,E1 -29898.548,E2 -29898.548} C_VEL
LIN {X 0,Y 60.76,Z 477.671,A -85,B 0,C 180,E1 -29902.711,E2 -29902.711} C_VEL
LIN {X 0,Y 59.078,Z 477.788,A -85,B 0,C 180,E1 -29905.993,E2 -29905.993} C_VEL
LIN {X 0,Y 55.455,Z 477.525,A -85,B 0,C 180,E1 -29911.935,E2 -29911.935} C_VEL
LIN {X 0,Y 50.434,Z 476.284,A -85,B 0,C 180,E1 -29920.287,E2 -29920.287} C_VEL
LIN {X 0,Y 49.163,Z 475.767,A -85,B 0,C 180,E1 -29922.464,E2 -29922.464} C_VEL
LIN {X 0,Y 42.893,Z 471.719,A -85,B 0,C 180,E1 -29940.558,E2 -29940.558} C_VEL
LIN {X 0,Y 41.913,Z 468.019,A -85,B 0,C 180,E1 -29955.433,E2 -29955.433} C_VEL
LIN {X 0,Y 42.141,Z 466.579,A -85,B 0,C 180,E1 -29960.4,E2 -29960.4} C_VEL
LIN {X 0,Y 40.97,Z 463.152,A -85,B 0,C 180,E1 -29967.542,E2 -29967.542} C_VEL
LIN {X 0,Y 40.037,Z 456.304,A -85,B 0,C 180,E1 -29980.11,E2 -29980.11} C_VEL
LIN {X 0,Y 39.277,Z 449.856,A -85,B 0,C 180,E1 -29989.603,E2 -29989.603} C_VEL
LIN {X 0,Y 39.086,Z 441.164,A -85,B 0,C 180,E1 -30000.647,E2 -30000.647} C_VEL
LIN {X 0,Y 39.989,Z 431.055,A -85,B 0,C 180,E1 -30011.227,E2 -30011.227} C_VEL
LIN {X 0,Y 41.696,Z 419.556,A -85,B 0,C 180,E1 -30020.479,E2 -30020.479} C_VEL
LIN {X 0,Y 43.616,Z 408.055,A -85,B 0,C 180,E1 -30027.401,E2 -30027.401} C_VEL
LIN {X 0,Y 42.491,Z 402.534,A -85,B 0,C 180,E1 -30031.606,E2 -30031.606} C_VEL
LIN {X 0,Y 38.434,Z 394.254,A -85,B 0,C 180,E1 -30040.915,E2 -30040.915} C_VEL
LIN {X 0,Y 37.213,Z 391.294,A -85,B 0,C 180,E1 -30045.115,E2 -30045.115} C_VEL
LIN {X 0,Y 37.283,Z 390.825,A -85,B 0,C 180,E1 -30049.134,E2 -30049.134} C_VEL
LIN {X 0,Y 37.981,Z 390.751,A -85,B 0,C 180,E1 -30060,E2 -30060} C_VEL
LIN {X 0,Y 37.334,Z 390.83,A -85,B 0,C 180,E1 -30070.85,E2 -30070.85} C_VEL
LIN {X 0,Y 37.056,Z 390.867,A -85,B 0,C 180,E1 -30078.512,E2 -30078.512} C_VEL
LIN {X 0,Y 36.725,Z 390.908,A -85,B 0,C 180,E1 -30095.037,E2 -30095.037} C_VEL
LIN {X 0,Y 36.727,Z 390.903,A -85,B 0,C 180,E1 -30100.057,E2 -30100.057} C_VEL
LIN {X 0,Y 36.727,Z 390.909,A -85,B 0,C 180,E1 -30109.945,E2 -30109.945} C_VEL
LIN {X 0,Y 36.724,Z 390.901,A -85,B 0,C 180,E1 -30114.963,E2 -30114.963} C_VEL
LIN {X 0,Y 37.058,Z 390.859,A -85,B 0,C 180,E1 -30131.485,E2 -30131.485} C_VEL
LIN {X 0,Y 37.559,Z 391.021,A -85,B 0,C 180,E1 -30142.609,E2 -30142.609} C_VEL
LIN {X 0,Y 38.196,Z 392.697,A -85,B 0,C 180,E1 -30146.044,E2 -30146.044} C_VEL
LIN {X 0,Y 40.189,Z 396.403,A -85,B 0,C 180,E1 -30151.253,E2 -30151.253} C_VEL
LIN {X 0,Y 42.219,Z 403.395,A -85,B 0,C 180,E1 -30158.375,E2 -30158.375} C_VEL
LIN {X 0,Y 44.071,Z 411.774,A -85,B 0,C 180,E1 -30166.202,E2 -30166.202} C_VEL
LIN {X 0,Y 45.453,Z 418.8,A -85,B 0,C 180,E1 -30172.735,E2 -30172.735} C_VEL
LIN {X 0,Y 42.245,Z 428.152,A -85,B 0,C 180,E1 -30180.626,E2 -30180.626} C_VEL
LIN {X 0,Y 38.882,Z 439.266,A -85,B 0,C 180,E1 -30193.697,E2 -30193.697} C_VEL
LIN {X 0,Y 37.588,Z 448.962,A -85,B 0,C 180,E1 -30209.061,E2 -30209.061} C_VEL
LIN {X 0,Y 39.263,Z 458.38,A -85,B 0,C 180,E1 -30227.071,E2 -30227.071} C_VEL
LIN {X 0,Y 45.323,Z 467.177,A -85,B 0,C 180,E1 -30244.447,E2 -30244.447} C_VEL
LIN {X 0,Y 53.097,Z 473.311,A -85,B 0,C 180,E1 -30255.351,E2 -30255.351} C_VEL
LIN {X 0,Y 63.119,Z 478.628,A -85,B 0,C 180,E1 -30263.89,E2 -30263.89} C_VEL
LIN {X 0,Y 65.555,Z 479.65,A -85,B 0,C 180,E1 -30265.394,E2 -30265.394} C_VEL
LIN {X 0,Y 52.799,Z 477.06,A -85,B 0,C 180,E1 -30277,E2 -30277} C_VEL
LIN {X 0,Y 49.163,Z 475.767,A -85,B 0,C 180,E1 -30282.464,E2 -30282.464} C_VEL
LIN {X 0,Y 45.798,Z 474.207,A -85,B 0,C 180,E1 -30288.005,E2 -30288.005} C_VEL
LIN {X 0,Y 40.269,Z 470.522,A -85,B 0,C 180,E1 -30297.781,E2 -30297.781} C_VEL
LIN {X 0,Y 36.866,Z 467.021,A -85,B 0,C 180,E1 -30307.19,E2 -30307.19} C_VEL
LIN {X 0,Y 35.648,Z 463.523,A -85,B 0,C 180,E1 -30318.328,E2 -30318.328} C_VEL
LIN {X 0,Y 33.548,Z 456.9,A -85,B 0,C 180,E1 -30333.002,E2 -30333.002} C_VEL
LIN {X 0,Y 33.168,Z 453.841,A -85,B 0,C 180,E1 -30339.144,E2 -30339.144} C_VEL
LIN {X 0,Y 32.034,Z 444.858,A -85,B 0,C 180,E1 -30354.29,E2 -30354.29} C_VEL
LIN {X 0,Y 32.516,Z 434.721,A -85,B 0,C 180,E1 -30368.611,E2 -30368.611} C_VEL
LIN {X 0,Y 34.517,Z 422.363,A -85,B 0,C 180,E1 -30381.75,E2 -30381.75} C_VEL
LIN {X 0,Y 36.925,Z 410.459,A -85,B 0,C 180,E1 -30390.811,E2 -30390.811} C_VEL
LIN {X 0,Y 37.094,Z 409.117,A -85,B 0,C 180,E1 -30391.727,E2 -30391.727} C_VEL
LIN {X 0,Y 36.307,Z 405.116,A -85,B 0,C 180,E1 -30395.711,E2 -30395.711} C_VEL
LIN {X 0,Y 32.666,Z 396.868,A -85,B 0,C 180,E1 -30407.575,E2 -30407.575} C_VEL
LIN {X 0,Y 30.678,Z 392.576,A -85,B 0,C 180,E1 -30416.305,E2 -30416.305} C_VEL
LIN {X 0,Y 30.81,Z 391.66,A -85,B 0,C 180,E1 -30420,E2 -30420} C_VEL
LIN {X 0,Y 30.109,Z 391.635,A -85,B 0,C 180,E1 -30433.498,E2 -30433.498} C_VEL
LIN {X 0,Y 29.864,Z 391.64,A -85,B 0,C 180,E1 -30439.73,E2 -30439.73} C_VEL
LIN {X 0,Y 29.496,Z 391.661,A -85,B 0,C 180,E1 -30448.459,E2 -30448.459} C_VEL
LIN {X 0,Y 29.542,Z 391.669,A -85,B 0,C 180,E1 -30465.536,E2 -30465.536} C_VEL
LIN {X 0,Y 29.595,Z 391.798,A -85,B 0,C 180,E1 -30485.061,E2 -30485.061} C_VEL
LIN {X 0,Y 30.063,Z 392.642,A -85,B 0,C 180,E1 -30490.363,E2 -30490.363} C_VEL
LIN {X 0,Y 31.539,Z 395.15,A -85,B 0,C 180,E1 -30497.125,E2 -30497.125} C_VEL
LIN {X 0,Y 32.83,Z 396.253,A -85,B 0,C 180,E1 -30500.761,E2 -30500.761} C_VEL
LIN {X 0,Y 34.541,Z 399.814,A -85,B 0,C 180,E1 -30507.084,E2 -30507.084} C_VEL
LIN {X 0,Y 35.96,Z 405.406,A -85,B 0,C 180,E1 -30514.203,E2 -30514.203} C_VEL
LIN {X 0,Y 37.73,Z 415.162,A -85,B 0,C 180,E1 -30525.254,E2 -30525.254} C_VEL
LIN {X 0,Y 38.452,Z 419.697,A -85,B 0,C 180,E1 -30530.307,E2 -30530.307} C_VEL
LIN {X 0,Y 34.187,Z 431.082,A -85,B 0,C 180,E1 -30542.005,E2 -30542.005} C_VEL
LIN {X 0,Y 31.028,Z 442.408,A -85,B 0,C 180,E1 -30559.369,E2 -30559.369} C_VEL
LIN {X 0,Y 30.829,Z 451.249,A -85,B 0,C 180,E1 -30577.571,E2 -30577.571} C_VEL
LIN {X 0,Y 34.346,Z 460.051,A -85,B 0,C 180,E1 -30597.364,E2 -30597.364} C_VEL
LIN {X 0,Y 41.988,Z 468.305,A -85,B 0,C 180,E1 -30613.807,E2 -30613.807} C_VEL
LIN {X 0,Y 51.497,Z 474.658,A -85,B 0,C 180,E1 -30624.169,E2 -30624.169} C_VEL
LIN {X 0,Y 53.075,Z 475.492,A -85,B 0,C 180,E1 -30625.399,E2 -30625.399} C_VEL
LIN {X 0,Y 50.838,Z 475.172,A -85,B 0,C 180,E1 -30628.74,E2 -30628.74} C_VEL
LIN {X 0,Y 41.202,Z 471.693,A -85,B 0,C 180,E1 -30643.024,E2 -30643.024} C_VEL
LIN {X 0,Y 35.832,Z 466.418,A -85,B 0,C 180,E1 -30666.904,E2 -30666.904} C_VEL
LIN {X 0,Y 35.648,Z 463.523,A -85,B 0,C 180,E1 -30678.328,E2 -30678.328} C_VEL
LIN {X 0,Y 35.29,Z 461.614,A -85,B 0,C 180,E1 -30683.548,E2 -30683.548} C_VEL
LIN {X 0,Y 34.193,Z 459.273,A -85,B 0,C 180,E1 -30688.187,E2 -30688.187} C_VEL
LIN {X 0,Y 31.708,Z 455.306,A -85,B 0,C 180,E1 -30694.611,E2 -30694.611} C_VEL
LIN {X 0,Y 25.484,Z 444.711,A -85,B 0,C 180,E1 -30711.895,E2 -30711.895} C_VEL
LIN {X 0,Y 24.931,Z 441.428,A -85,B 0,C 180,E1 -30718.042,E2 -30718.042} C_VEL
LIN {X 0,Y 25.977,Z 431.262,A -85,B 0,C 180,E1 -30735.249,E2 -30735.249} C_VEL
LIN {X 0,Y 28.766,Z 418.944,A -85,B 0,C 180,E1 -30750.096,E2 -30750.096} C_VEL
LIN {X 0,Y 30.656,Z 411.411,A -85,B 0,C 180,E1 -30756.49,E2 -30756.49} C_VEL
LIN {X 0,Y 30.649,Z 408.919,A -85,B 0,C 180,E1 -30759.18,E2 -30759.18} C_VEL
LIN {X 0,Y 27.894,Z 401.403,A -85,B 0,C 180,E1 -30772.755,E2 -30772.755} C_VEL
LIN {X 0,Y 26.73,Z 398.572,A -85,B 0,C 180,E1 -30779.999,E2 -30779.999} C_VEL
LIN {X 0,Y 25.479,Z 396.964,A -85,B 0,C 180,E1 -30787.927,E2 -30787.927} C_VEL
LIN {X 0,Y 24.345,Z 396.032,A -85,B 0,C 180,E1 -30796.779,E2 -30796.779} C_VEL
LIN {X 0,Y 23.607,Z 395.565,A -85,B 0,C 180,E1 -30806.736,E2 -30806.736} C_VEL
LIN {X 0,Y 23.379,Z 395.67,A -85,B 0,C 180,E1 -30816.956,E2 -30816.956} C_VEL
LIN {X 0,Y 24.821,Z 397.185,A -85,B 0,C 180,E1 -30838.149,E2 -30838.149} C_VEL
LIN {X 0,Y 26.168,Z 398.282,A -85,B 0,C 180,E1 -30846.537,E2 -30846.537} C_VEL
LIN {X 0,Y 28.593,Z 402.331,A -85,B 0,C 180,E1 -30859.473,E2 -30859.473} C_VEL
LIN {X 0,Y 29.458,Z 405.15,A -85,B 0,C 180,E1 -30864.862,E2 -30864.862} C_VEL
LIN {X 0,Y 30.43,Z 411.307,A -85,B 0,C 180,E1 -30873.937,E2 -30873.937} C_VEL
LIN {X 0,Y 31.414,Z 419.001,A -85,B 0,C 180,E1 -30884.743,E2 -30884.743} C_VEL
LIN {X 0,Y 31.301,Z 420.927,A -85,B 0,C 180,E1 -30887.08,E2 -30887.08} C_VEL
LIN {X 0,Y 26.495,Z 432.688,A -85,B 0,C 180,E1 -30902.039,E2 -30902.039} C_VEL
LIN {X 0,Y 23.778,Z 443.286,A -85,B 0,C 180,E1 -30923.764,E2 -30923.764} C_VEL
LIN {X 0,Y 24.748,Z 452.354,A -85,B 0,C 180,E1 -30947.703,E2 -30947.703} C_VEL
LIN {X 0,Y 30.832,Z 461.734,A -85,B 0,C 180,E1 -30970.648,E2 -30970.648} C_VEL
LIN {X 0,Y 40.594,Z 469.786,A -85,B 0,C 180,E1 -30985.125,E2 -30985.125} C_VEL
LIN {X 0,Y 42.464,Z 470.98,A -85,B 0,C 180,E1 -30986.892,E2 -30986.892} C_VEL
LIN {X 0,Y 33.774,Z 467.196,A -85,B 0,C 180,E1 -31003.257,E2 -31003.257} C_VEL
LIN {X 0,Y 29.505,Z 461.188,A -85,B 0,C 180,E1 -31032.325,E2 -31032.325} C_VEL
LIN {X 0,Y 28.429,Z 458.842,A -85,B 0,C 180,E1 -31038.951,E2 -31038.951} C_VEL
LIN {X 0,Y 26.634,Z 453.009,A -85,B 0,C 180,E1 -31053.782,E2 -31053.782} C_VEL
LIN {X 0,Y 25.107,Z 445.239,A -85,B 0,C 180,E1 -31070.48,E2 -31070.48} C_VEL
LIN {X 0,Y 24.931,Z 441.428,A -85,B 0,C 180,E1 -31078.042,E2 -31078.042} C_VEL
LIN {X 0,Y 24.476,Z 436.826,A -85,B 0,C 180,E1 -31086.438,E2 -31086.438} C_VEL
LIN {X 0,Y 22.993,Z 428.947,A -85,B 0,C 180,E1 -31100.659,E2 -31100.659} C_VEL
LIN {X 0,Y 22.637,Z 420.755,A -85,B 0,C 180,E1 -31114.932,E2 -31114.932} C_VEL
LIN {X 0,Y 23.728,Z 415.558,A -85,B 0,C 180,E1 -31121.605,E2 -31121.605} C_VEL
LIN {X 0,Y 24.742,Z 412.357,A -85,B 0,C 180,E1 -31124.659,E2 -31124.659} C_VEL
LIN {X 0,Y 24.337,Z 410.336,A -85,B 0,C 180,E1 -31128.651,E2 -31128.651} C_VEL
LIN {X 0,Y 23.244,Z 405.785,A -85,B 0,C 180,E1 -31139.999,E2 -31139.999} C_VEL
LIN {X 0,Y 22.892,Z 404.391,A -85,B 0,C 180,E1 -31144.406,E2 -31144.406} C_VEL
LIN {X 0,Y 21.791,Z 402.834,A -85,B 0,C 180,E1 -31154.636,E2 -31154.636} C_VEL
LIN {X 0,Y 21.406,Z 402.476,A -85,B 0,C 180,E1 -31159.166,E2 -31159.166} C_VEL
LIN {X 0,Y 20.764,Z 402.638,A -85,B 0,C 180,E1 -31182.604,E2 -31182.604} C_VEL
LIN {X 0,Y 22.023,Z 403.839,A -85,B 0,C 180,E1 -31199.494,E2 -31199.494} C_VEL
LIN {X 0,Y 23.894,Z 407.555,A -85,B 0,C 180,E1 -31215.849,E2 -31215.849} C_VEL
LIN {X 0,Y 24.249,Z 411.396,A -85,B 0,C 180,E1 -31223.754,E2 -31223.754} C_VEL
LIN {X 0,Y 24.711,Z 419.139,A -85,B 0,C 180,E1 -31237.73,E2 -31237.73} C_VEL
LIN {X 0,Y 24.815,Z 420.779,A -85,B 0,C 180,E1 -31240.585,E2 -31240.585} C_VEL
LIN {X 0,Y 19.736,Z 431.738,A -85,B 0,C 180,E1 -31257.097,E2 -31257.097} C_VEL
LIN {X 0,Y 16.787,Z 442.585,A -85,B 0,C 180,E1 -31286.857,E2 -31286.857} C_VEL
LIN {X 0,Y 19.185,Z 452.271,A -85,B 0,C 180,E1 -31320.001,E2 -31320.001} C_VEL
LIN {X 0,Y 27.13,Z 461.406,A -85,B 0,C 180,E1 -31342.866,E2 -31342.866} C_VEL
LIN {X 0,Y 31.508,Z 464.965,A -85,B 0,C 180,E1 -31348.9,E2 -31348.9} C_VEL
LIN {X 0,Y 30.304,Z 464.498,A -85,B 0,C 180,E1 -31352.736,E2 -31352.736} C_VEL
LIN {X 0,Y 23.952,Z 458.995,A -85,B 0,C 180,E1 -31381.675,E2 -31381.675} C_VEL
LIN {X 0,Y 23.445,Z 457.771,A -85,B 0,C 180,E1 -31387.535,E2 -31387.535} C_VEL
LIN {X 0,Y 20.501,Z 452.003,A -85,B 0,C 180,E1 -31405.079,E2 -31405.079} C_VEL
LIN {X 0,Y 18.367,Z 445.375,A -85,B 0,C 180,E1 -31423.836,E2 -31423.836} C_VEL
LIN {X 0,Y 18.482,Z 434.163,A -85,B 0,C 180,E1 -31452.879,E2 -31452.879} C_VEL
LIN {X 0,Y 21.547,Z 422.366,A -85,B 0,C 180,E1 -31473.759,E2 -31473.759} C_VEL
LIN {X 0,Y 23.728,Z 415.558,A -85,B 0,C 180,E1 -31481.605,E2 -31481.605} C_VEL
LIN {X 0,Y 23.506,Z 414.158,A -85,B 0,C 180,E1 -31484.382,E2 -31484.382} C_VEL
LIN {X 0,Y 21.681,Z 412.99,A -85,B 0,C 180,E1 -31491.128,E2 -31491.128} C_VEL
LIN {X 0,Y 19.206,Z 411.832,A -85,B 0,C 180,E1 -31503.147,E2 -31503.147} C_VEL
LIN {X 0,Y 18.959,Z 411.089,A -85,B 0,C 180,E1 -31506.564,E2 -31506.564} C_VEL
LIN {X 0,Y 18.899,Z 409.917,A -85,B 0,C 180,E1 -31510.726,E2 -31510.726} C_VEL
LIN {X 0,Y 18.071,Z 408.986,A -85,B 0,C 180,E1 -31522.885,E2 -31522.885} C_VEL
LIN {X 0,Y 17.651,Z 409.048,A -85,B 0,C 180,E1 -31537.219,E2 -31537.219} C_VEL
LIN {X 0,Y 18.076,Z 409.592,A -85,B 0,C 180,E1 -31551.042,E2 -31551.042} C_VEL
LIN {X 0,Y 18.574,Z 410.491,A -85,B 0,C 180,E1 -31559.66,E2 -31559.66} C_VEL
LIN {X 0,Y 19.096,Z 412.076,A -85,B 0,C 180,E1 -31568.406,E2 -31568.406} C_VEL
LIN {X 0,Y 18.527,Z 419.245,A -85,B 0,C 180,E1 -31585.917,E2 -31585.917} C_VEL
LIN {X 0,Y 18.463,Z 420.916,A -85,B 0,C 180,E1 -31590,E2 -31590} C_VEL
LIN {X 0,Y 18.085,Z 422.028,A -85,B 0,C 180,E1 -31591.841,E2 -31591.841} C_VEL
LIN {X 0,Y 12.176,Z 432.912,A -85,B 0,C 180,E1 -31613.615,E2 -31613.615} C_VEL
LIN {X 0,Y 10.03,Z 442.743,A -85,B 0,C 180,E1 -31659.492,E2 -31659.492} C_VEL
LIN {X 0,Y 16.76,Z 453.698,A -85,B 0,C 180,E1 -31704.794,E2 -31704.794} C_VEL
